(* CODESYS project DemoNov3.project
   Author: Cooper Power Systems
   Title: CoDeSys Project
   Version: 1.0.0.0
   Description: Sample Project
   Company: Cooper Power Systems LLC

Project tree, tasks and I/O mapping:
  Device : SMP SG 4000, Cooper Power Systems, LLC., order no. 
      , version 3.5.2.0
    application Application
      libraries: SmpLib, 3.5.2.0 (Cooper Power Systems); Standard, 3.5.2.0 (System)
      task Main_Task (cyclic, interval T#10ms, priority 0) calls PLC_MAIN, Tasks_10ms
      task Task_50ms (cyclic, interval t#250ms, priority 1) calls Tasks_50ms
      task Task_100ms (cyclic, interval t#100ms, priority 2) calls Tasks_100ms
      task Task_300ms (cyclic, interval t#250ms, priority 2) calls Task_300ms, POU_EXPORT
      global variables PersistentVars
      POUs/
        program PLC_MAIN [ST]
        program POU_EXPORT [ST]
        program SMP_Csys_var_AI [ST]
        program MICROGRID_MODES [ST]
        program VDC [ST]
        program SMP_Csys_var_AO [FBD]
        program LOAD_Balance [ST]
        program Load_Shed [ST]
        program SMP_OUTPUTS [FBD]
        program INIT [ST]
        program Vijay [FBD]
        program Timers [FBD]
        program PCC_CNTL [FBD]
        program Tasks_10ms [ST]
        program MICROGRID_Apps [ST]
        program Tasks_50ms [ST]
        program Tasks_100ms [ST]
        program Task_300ms [ST]
        program BRK_CNTL [ST]
        program POU_RESET [ST]
        program SMP_AO [ST]
        program TIMER_ST [ST]
        program PCC_PROTECT [ST]
        program SOC_MNGT [ST]
        program Q_Export [ST]
      function block SMP_MAP_SYMBOLS [ST]
      global variables SMP_global_symbols_declaration
      global variables Global_Variables
  function GetNumberProperty [ST]
  function GetBooleanProperty [ST]
  function GetCompany [ST]
  function GetTitle [ST]
  function GetVersionProperty [ST]
  function GetVersion [ST]
  function GetTextProperty [ST]
*)

// Device/Application/PersistentVars
VAR_GLOBAL PERSISTENT RETAIN
	PERSIST_COUNTER: DINT := 0;
	CONDITION: INT;
	GRID_APP_SELECT: INT := 0;
	ISLAND_APP_SELECT: INT := 0;
	
	// Lower frequency power limit for G1
	F_G1_L: REAL := 0;
	F_G1_H: REAL := 0;
	F_G2_L: REAL := 0;
	F_G2_H: REAL := 0;
	F_PV_L: REAL := 0;
	F_PV_H: REAL := 0;
	F_ES_L: REAL := 0;
	F_ES_H: REAL := 0;
	
	F_L9_L: REAL := 0;
	F_L9_H: REAL := 0;
	F_L10_L: REAL := 0;
	F_L10_H: REAL := 0;
	F_L11_L: REAL := 0;
	F_L11_H: REAL := 0;
	F_L15_L: REAL := 0;
	F_L15_H: REAL := 0;
	F_L16_L: REAL := 0;
	F_L16_H: REAL := 0;
	F_L20_L: REAL := 0;
	F_L20_H: REAL := 0;
	
	P_R2: REAL := 0;
	P_R3: REAL := 0;
	P_R4: REAL := 0;
	P_R5: REAL := 0;
	P_R6: REAL := 0;
	P_R7: REAL := 0;
	P_R8: REAL := 0;
	P_R9: REAL := 0;
	P_R10: REAL := 0;
	P_R11: REAL := 0;
	P_R12: REAL := 0;
	P_R13: REAL := 0;
	P_R14: REAL := 0;
	P_R15: REAL := 0;
	P_R16: REAL := 0;
	P_R17: REAL := 0;
	P_R18: REAL := 0;
	P_R19: REAL := 0;
	P_R20: REAL := 0;
	P_R21: REAL := 0;
	P_R22: REAL := 0;
	Q_R2: REAL := 0;
	Q_R3: REAL := 0;
	Q_R4: REAL := 0;
	Q_R5: REAL := 0;
	Q_R6: REAL := 0;
	Q_R7: REAL := 0;
	Q_R8: REAL := 0;
	Q_R9: REAL := 0;
	Q_R10: REAL := 0;
	Q_R11: REAL := 0;
	Q_R12: REAL := 0;
	Q_R13: REAL := 0;
	Q_R14: REAL := 0;
	Q_R15: REAL := 0;
	Q_R16: REAL := 0;
	Q_R17: REAL := 0;
	Q_R18: REAL := 0;
	Q_R19: REAL := 0;
	Q_R20: REAL := 0;
	Q_R21: REAL := 0;
	Q_R22: REAL := 0;
	StPCC: INT := 0;
	PTL_Mode1: REAL := 0;
	PTL_Mode2: REAL := 0;
	QTL_Mode1: REAL := 0;
	QTL_Mode2: REAL := 0;
//	MG_Base_P: REAL := 9.0;
//	MG_Base_Q: REAL := 5.0;
	F_BL_L: REAL := 0;
	F_BL_H: REAL := 0;
	F: REAL := 0;
	Gen1_CapW: REAL := 0;
	V_G1_L: REAL := 0;
	V_G1_H: REAL := 0;
	V_G2_L: REAL := 0;
	V_G2_H: REAL := 0;
	V_PV_L: REAL := 0;
	V_PV_H: REAL := 0;
	V_ES_L: REAL := 0;
	V_ES_H: REAL := 0;
	
	V_L9_L: REAL := 0;
	V_L9_H: REAL := 0;
	V_L10_L: REAL := 0;
	V_L10_H: REAL := 0;
	V_L11_L: REAL := 0;
	V_L11_H: REAL := 0;
	V_L15_L: REAL := 0;
	V_L15_H: REAL := 0;
	V_L16_L: REAL := 0;
	V_L16_H: REAL := 0;
	V_L20_L: REAL := 0;
	V_L20_H: REAL := 0;

	V_BL_L: REAL := 0;
	V_BL_H: REAL := 0;
	V: REAL := 0;
	Gen1_Capkvar: REAL := 0;
	Gen2_CapW: REAL := 0;
	Gen2_Capkvar: REAL := 0;
	PESS_CMD: REAL := 0;
	QESS_CMD: REAL := 0;
	BRK_PCC_CNTL: INT := 0;
	BRK_O2_CNTL: INT := 0;
	BRK_O3_CNTL: INT := 0;
	BRK_O4_CNTL: INT := 0;
	BRK_O5_CNTL: INT := 0;
	BRK_O6_CNTL: INT := 0;
	BRK_O7_CNTL: INT := 0;
	BRK_O8_CNTL: INT := 0;
	BRK_O9_CNTL: INT := 0;
	BRK_O10_CNTL: INT := 0;
	BRK_O11_CNTL: INT := 0;
	BRK_O12_CNTL: INT := 0;
	BRK_O13_CNTL: INT := 0;
	BRK_O14_CNTL: INT := 0;
	BRK_O15_CNTL: INT := 0;
	BRK_O16_CNTL: INT := 0;
	BRK_O17_CNTL: INT := 0;
	BRK_O18_CNTL: INT := 0;
	BRK_O19_CNTL: INT := 0;
	BRK_O20_CNTL: INT := 0;
	BRK_O21_CNTL: INT := 0;
	BRK_O22_CNTL: INT := 0;
	// GEN1 start/stop command
	GEN1_SS_CNTL: INT := 0;
	GEN2_SS_CNTL: INT := 0;
	ESS_SS_CNTL: INT := 0;
	PV_SS_CNTL: INT := 0;
	GEN1_MOD_sel: INT := 0;
	GEN2_MOD_sel: INT := 0;
	BAT_Enb_set: INT := 0;
	//kw//
	GEN1_kW_Out: REAL := 0;
	MG_kW_Out: REAL := 0;
	GEN2_kW_Out: REAL := 0;
	ESS_kW_Out: REAL := 0;
	PV_kW_Out: REAL := 0;
	MG_kW_Bal: REAL := 0;
	
	//kvar//
	GEN1_kVAr_Out: REAL := 0;
	MG_kVAr_Out: REAL := 0;
	GEN2_kVAr_Out: REAL := 0;
	ESS_kVAr_Out: REAL := 0;
	PV_kVAr_Out: REAL := 0;
	MG_kVAr_Bal: REAL := 0;
	
	BRKGEN1_TRIG: BOOL := 0;
	BRKGEN1_RTRIG: R_TRIG;
	BRKGEN1_FTRIG: F_TRIG;
	
	BRKGEN2_TRIG: BOOL := 0;
	BRKGEN2_RTRIG: R_TRIG;
	BRKGEN2_FTRIG: F_TRIG;
	
	BRKESS_TRIG: BOOL := 0;
	BRKESS_RTRIG: R_TRIG;
	BRKESS_FTRIG: F_TRIG;
	
	BRKPCC_TRIG: BOOL := 0;
	BRKPCC_RTRIG: R_TRIG;
	BRKPCC_FTRIG: F_TRIG;
	
	BRK2_TRIG: BOOL := 0;
	BRK2_RTRIG: R_TRIG;
	BRK2_FTRIG: F_TRIG;
	BRK3_TRIG: BOOL := 0;
	BRK3_RTRIG: R_TRIG;
	BRK3_FTRIG: F_TRIG;
	BRK4_TRIG: BOOL := 0;
	BRK4_RTRIG: R_TRIG;
	BRK4_FTRIG: F_TRIG;
	BRK5_TRIG: BOOL := 0;
	BRK5_RTRIG: R_TRIG;
	BRK5_FTRIG: F_TRIG;
	BRK6_TRIG: BOOL := 0;
	BRK6_RTRIG: R_TRIG;
	BRK6_FTRIG: F_TRIG;
	BRK7_TRIG: BOOL := 0;
	BRK7_RTRIG: R_TRIG;
	BRK7_FTRIG: F_TRIG;
	BRK8_TRIG: BOOL := 0;
	BRK8_RTRIG: R_TRIG;
	BRK8_FTRIG: F_TRIG;
	BRK9_TRIG: BOOL := 0;
	BRK9_RTRIG: R_TRIG;
	BRK9_FTRIG: F_TRIG;
	BRK10_TRIG: BOOL := 0;
	BRK10_RTRIG: R_TRIG;
	BRK10_FTRIG: F_TRIG;
	BRK11_TRIG: BOOL := 0;
	BRK11_RTRIG: R_TRIG;
	BRK11_FTRIG: F_TRIG;
	BRK12_TRIG: BOOL := 0;
	BRK12_RTRIG: R_TRIG;
	BRK12_FTRIG: F_TRIG;
	BRK13_TRIG: BOOL := 0;
	BRK13_RTRIG: R_TRIG;
	BRK13_FTRIG: F_TRIG;
	BRK14_TRIG: BOOL := 0;
	BRK14_RTRIG: R_TRIG;
	BRK14_FTRIG: F_TRIG;
	BRK15_TRIG: BOOL := 0;
	BRK15_RTRIG: R_TRIG;
	BRK15_FTRIG: F_TRIG;
	BRK16_TRIG: BOOL := 0;
	BRK16_RTRIG: R_TRIG;
	BRK16_FTRIG: F_TRIG;
	BRK17_TRIG: BOOL := 0;
	BRK17_RTRIG: R_TRIG;
	BRK17_FTRIG: F_TRIG;
	BRK18_TRIG: BOOL := 0;
	BRK18_RTRIG: R_TRIG;
	BRK18_FTRIG: F_TRIG;
	BRK19_TRIG: BOOL := 0;
	BRK19_RTRIG: R_TRIG;
	BRK19_FTRIG: F_TRIG;
	BRK20_TRIG: BOOL := 0;
	BRK20_RTRIG: R_TRIG;
	BRK20_FTRIG: F_TRIG;
	BRK21_TRIG: BOOL := 0;
	BRK21_RTRIG: R_TRIG;
	BRK21_FTRIG: F_TRIG;
	BRK22_TRIG: BOOL := 0;
	BRK22_RTRIG: R_TRIG;
	BRK22_FTRIG: F_TRIG;
	PCC_BRK_ST2: R_TRIG;
	BRK_toggle: BOOL := 0;
	//Load Shed variables
	I_Load_02: INT := 0;//Not Used
	I_Load_03: INT := 0;//Not Used
	I_Load_04: INT := 0;//Not Used
	I_Load_05: INT := 0;
	I_Load_06: INT := 0;//Not Used
	I_Load_07: INT := 0;//Not Used
	I_Load_08: INT := 0;//Not Used
	I_Load_09: INT := 0;
	I_Load_10: INT := 0;
	I_Load_11: INT := 0;
	I_Load_012: INT := 0;//Not Used
	I_Load_013: INT := 0;//Not Used
	C_Load_014: INT := 0;
	I_Load_015: INT := 0;
	I_Load_016: INT := 0;
	I_Load_017: INT := 0;//Not Used
	C_Load_018: INT := 0;
	C_Load_019: INT := 0;
	C_Load_020: INT := 0;
	C_Load_021: INT := 0;
	C_Load_022: INT := 0;
	
	
	
	
	
	
	RESET_All: BOOL := 0;
	ISLAND_CMD: BOOL := 0;
	
	
	
	
	//Export
	ERR_T: REAL := 0;
	INT_ERR: REAL := 0;
	MG_kW_Bal2: REAL := 0;
	MG_kW_Bal3: REAL := 0;
	
	GEN2_ON: BOOL := 0;
	GEN1_ON: BOOL := 0;
	ESS_ON: BOOL := 0;
	BAT_CAP: REAL := 0;
	MSTRST2: TOF;
	PCC_Delay: TON;
END_VAR

// Device/Application/SMP_global_symbols_declaration
VAR_GLOBAL
	///
	///Consumed Ai
	SPS_ADAM1_ADAM_AI_3: AI_IN;
	SPS_ADAM1_ADAM_AI_5: AI_IN;
	SPS_GEN1_METMMXU1HzInstMag: AI_IN;
	SPS_GEN1_METMMXU1TotVArInstMag: AI_IN;
	SPS_GEN1_METMMXU1TotWInstMag: AI_IN;
	SPS_PCS_drv1_Iq_ref: AI_IN;
	SPS_SELG_METYMMXU2HzInstMag: AI_IN;
	SPS_SELG_METYMMXU2HzMag: AI_IN;
	SPS_SELG_METYMMXU2PhVPhsAIMag: AI_IN;
	SPS_SELG_METYMMXU2PhVPhsAMag: AI_IN;
	SPS_SELG_METYMMXU2TotVArInstMag: AI_IN;
	SPSSELG_METYMMXU2TotVArMag: AI_IN;
	SPSSELG_METYMMXU2TotWInstMag: AI_IN;
	SPS_SELG_METYMMXU2TotWMag: AI_IN;
	///
	///Consumed Ao
	SPS_PCS_INV1_FB2_POWDEL_INS: AO_IN;
	SPS_PCS_INV1_FB3_POWDEL_INS: AO_IN;
END_VAR

// Device/Application/Global_Variables
VAR_GLOBAL

	
PCC_BRK_ST: DINT := 0;    // 1 = BRK_Closed  0 = BRK_Open
	MIN_CLK: BOOL;
	HR_CLK: BOOL;
	Mode1_CNTR_flg: BOOL := 0;
	RUN_MIN: INT := 0;
	PPCC_CMD: REAL := 0;
	QPCC_CMD: REAL := 0;
	TMR_MIN_1: TON;
	Mode1_CNTR_1: CTU;
	TMR1_1: TON;
	TMRs_1: TON;
	Fretest: DINT := 0;
	AO_TGL_1: TON;
	AO_TGL_2: TON;
	EXP_CMD: BOOL := 0;
	Trig3: INT := 0;
	Trig4: BOOL := 0;
END_VAR
VAR_GLOBAL RETAIN
	Adam_UPC: CTU;
	T_2 : BOOL;
	T_1 : BOOL;
	ON_OFF_SW: INT;
	OUT_Visualisation: BOOL := 0;
	SET5: BOOL;
	B_Switch: BOOL := 0;
	DRV1_Cmd_Data: DINT := 0;
	DRV2_Cmd_Data: DINT := 0;
	Real_P1: DINT := 0;
	Real_P2: DINT := 0;
	SPS_Rreal_Pw: DINT := 0;
	React_P1: DINT := 0;
	React_P2: DINT := 0;
	SPS_Reactive_Pw: DINT := 0;
	PTL: REAL := 0;
	QTL: REAL := 0;
	PT: REAL := 0;
	QT: REAL := 0;
	CPG1: REAL := 10;
	CPG2: REAL := 20;
	PG1_CMD: REAL;
	PG2_CMD: REAL := 0;
	
	QG1_CMD: REAL := 0;
	QG2_CMD: REAL := 0;
	
	QG1_CMD_A: REAL := 0;
	QG2_CMD_A: REAL := 0;
	
	QG1_CMD_B: REAL := 0;
	QG2_CMD_B: REAL := 0;
	
	
	CQG1: REAL := 10;
	CQG2: REAL := 20;
	MODE: INT := 0;
	MSTRST: R_TRIG;
	Trig: BOOL := 1;
	Load_Cntr: INT := 0;
	GEN1_toggle: BOOL := 0;
	GEN2_toggle: BOOL := 0;
	ESS_toggle: BOOL := 0;
	
	///Timing
	EXP_STRT1 : INT := 5;
	EXP_STRT2 : INT := 20;
	EXP_END : INT := 35;
	ISL_STRT : INT := 36;
	ISL_END : INT := 50;
	
	MG_Base_P: REAL := 9.0;
	MG_Base_Q: REAL := 5.0;
	
END_VAR

// Device/Application/POUs/PLC_MAIN
PROGRAM PLC_MAIN

VAR
	CODESYS_INIT: BOOL := FALSE;
	CODESYS_MAP: BOOL := FALSE;
	SmpMapSymbols : SMP_MAP_SYMBOLS;
	test: INT := 0;
	test1: INT := 0;
END_VAR

(* 	Cooper Power Systems LLC
	SoftPLC Sample project
	Version 1.0, January 2013
	
	This sample is provided "as is" to reduce the user's learning curve about CoDeSys integration with the SMP Gateway. 
	Cooper Power Systems cannot be held responsible in any situation resulting from the use of this sample program.

	Currently, the SMP Gateway runtime can only run one application at a time.
    This application must be named "Application".
	This application can be developped in any IEC 611l31-3 language.

	------------- IMPORTANT (begin)------------- 
	SMP Config automatically generates a PLCopenXML file that contains the SMP_MAP_SYMBOLS function block
    and the SMP_global_symbols_declaration global variable list. When the configuration of the SoftPLC component is changed in
    SMP Config, the content of this file must then be used to update the application.

	
	To update the application with the latest version of the PLCopenXML file, follow those steps:
	
	1. In the left pane, expand the project tree and select the "Application" branch under "PLC Logic".
	2. From the "Project" menu, choose "Import PLCopenXML"
	3. Select the XML file created by SMP Config. 
		The file is under My Documents or Documents/SMP Manager/Config Files/CoDeSys_TmpEdit. 
		The filename syntax is: the SMP Config settings filename + the Soft PLC instance name + "PLCopenXML.xml".
	4.  In the "Import PLCopenXML" window, just click "Open"; the two SMP-Gateway-related items are already selected.
	5. In the next window, select option 4 "Replace the existing object. Do the same for all subsequent conflicts."
	6. You ready to rebuild the application. 

	------------- IMPORTANT (end)------------- 
*)

(* 	The code inside this IF block must be executed first, ONLY once. *)
IF (SMF_CANMAPPLC(0) AND CODESYS_INIT = FALSE) THEN

	(*  Specify basic information about this application.
		Update according to your own application requirements and functionalities. *)
	SMF_INITPLC ('Application Name is Sample',  'Author is Cooper Power Systems, LLC', 'Description is a sample program',  '1.0', LIBVERSION, T#10S);

	(* 	Add a log entry indicating that the application is starting up.
		Update as required; you can also add additional SMF_LOG function call if you want *)
	SMF_LOG(TRUE, LOG_STARTUP,'SoftPLC application is starting');
	
	(* 	SMP_Config auto-generated symbol mapping.
	   	At runtime, an exception will be thrown if there is an error. 
	   	Use SMP Log and SMP Stats to get details about the error. 
		DO NOT DELETE THIS FUNCTION CALL. *)
	SmpMapSymbols();
			
	(* 	Update the initialization flag to indicates that initialization is complete.
		DO NOT DELETE THIS LINE OF CODE. *)
	CODESYS_INIT:=TRUE;
	//INIT();	
	test := test+1;
	
ELSE
	(* The code inside this IF block must be executed ONLY once, when the symbol mapping was successful. *)
	IF (SMF_CANSTARTPLC(0) AND CODESYS_MAP = FALSE) THEN
	
		(*  Initialize the output points synbols so they can accept control requests. 	
			Change/update as required. *)
		//( B:=0, Q:=0, DIS:= FALSE, END:=FALSE );
		//( I:= 0, Q:=0, DIS:= FALSE, END:=FALSE );
		//( F:= 0.0, Q:=0 );
			
		(* 	Examples on how to write an entry into each different log.
			Change/update as required. *) 
		SMF_LOG(TRUE, LOG_APPLICATION, 'Application Log: Example PLC');
		SMF_LOG(TRUE, LOG_COMMAND,'Control Log: Example PLC');
		SMF_LOG(TRUE, LOG_FILE,'File Log: Example PLC');
		SMF_LOG(TRUE, LOG_PROTOCOL,'Protocol Log: Example PLC');
		SMF_LOG(TRUE, LOG_SECURITY,'Security Log: Example PLC');
	
		(* 	Examples on how to write to each statistic field.
			Change/update as required. *)
		SMF_STAT(TRUE, STAT_USER1, '0'); 	(* BO CMND counter *)
		SMF_STAT(TRUE, STAT_USER2, '0'); 	(* AO CMND counter *)
		SMF_STAT(TRUE, STAT_USER3, 'No Used');
		SMF_STAT(TRUE, STAT_USER4, 'No Used');
		SMF_STAT(TRUE, STAT_USER5, 'No Used');
		SMF_STAT(TRUE, STAT_USER6, 'No Used');
		SMF_STAT(TRUE, STAT_USER7, 'No Used');
		SMF_STAT(TRUE, STAT_USER8, 'No Used');
		SMF_STAT(TRUE, STAT_USER9, 'No Used');
		SMF_STAT(TRUE, STAT_USER10, 'No Used');
		SMF_STAT(TRUE, STAT_USER11, 'No Used');
		SMF_STAT(TRUE, STAT_USER12, 'No Used');
		SMF_STAT(TRUE, STAT_USER13, 'No Used');
		SMF_STAT(TRUE, STAT_USER14, 'No Used');
		SMF_STAT(TRUE, STAT_USER15, 'No Used');
		SMF_STAT(TRUE, STAT_USER16, 'No Used');
	
		(* 	Add a log entry to indicate that the SoftPLC application was started successfully.
			Change/update as required. *)
		SMF_LOG(TRUE, LOG_STARTUP,'SoftPLC application is started.');
	
		(* 	Always re-enable local control operation
			This is specific to sample project: REMOVE IT FROM YOUR OWN APPLICATION *)	
		//( CMD:=BO_CMD_OPEN , ON:=T#0S , OFF:=T#0S , RPT:=0 , OP:=1 );
		//INPUT_BO_SetLocalControl( OP:=0 );
		
		(* 	Symbol mapping is completed and all points were initialized.
			DO NOT DELETE THIS LINE OF CODE. *)
		CODESYS_MAP:=TRUE;
	
	(* The code inside this IF block must be executed at each cycle, once INIT is completed. *)
	ELSIF (SMF_CANSTARTPLC(0) AND CODESYS_MAP = TRUE) THEN
	
		(* 	Call the main application coded in Structured Text.
			You can call any of your programs coded in any IEC 61131-3 language here.
			Change/update as required. *)
	//	ST_PROGRAM();
	//	Vijay();
	//	Timers();
		IF MSTRST2.Q = 1 THEN
			POU_RESET();
			test1 := test1+1;
		END_IF
	END_IF
END_IF

END_PROGRAM

// Device/Application/SMP_MAP_SYMBOLS
FUNCTION_BLOCK SMP_MAP_SYMBOLS

	(* Auto-generated by SMP Config, do not modify *)

	(* Subscribed points mapping *)
	SMF_MAP_AI_IN(ADR(SPS_ADAM1_ADAM_AI_3), 'ADAM1_ADAM_AI_3', 0);
	SMF_MAP_AI_IN(ADR(SPS_ADAM1_ADAM_AI_5), 'ADAM1_ADAM_AI_5', 0);
	SMF_MAP_AI_IN(ADR(SPS_GEN1_METMMXU1HzInstMag), 'GEN1_METMMXU1HzInstMag', 0);
	SMF_MAP_AI_IN(ADR(SPS_GEN1_METMMXU1TotVArInstMag), 'GEN1_METMMXU1TotVArInstMag', 0);
	SMF_MAP_AI_IN(ADR(SPS_GEN1_METMMXU1TotWInstMag), 'GEN1_METMMXU1TotWInstMag', 0);
	SMF_MAP_AI_IN(ADR(SPS_PCS_drv1_Iq_ref), 'PCS_drv1_Iq_ref', 0);
	SMF_MAP_AI_IN(ADR(SPS_SELG_METYMMXU2HzInstMag), 'SELG_METYMMXU2HzInstMag', 0);
	SMF_MAP_AI_IN(ADR(SPS_SELG_METYMMXU2HzMag), 'SELG_METYMMXU2HzMag', 0);
	SMF_MAP_AI_IN(ADR(SPS_SELG_METYMMXU2PhVPhsAIMag), 'SELG_METYMMXU2PhVPhsAIMag', 0);
	SMF_MAP_AI_IN(ADR(SPS_SELG_METYMMXU2PhVPhsAMag), 'SELG_METYMMXU2PhVPhsAMag', 0);
	SMF_MAP_AI_IN(ADR(SPS_SELG_METYMMXU2TotVArInstMag), 'SELG_METYMMXU2TotVArInstMag', 0);
	SMF_MAP_AI_IN(ADR(SPSSELG_METYMMXU2TotVArMag), 'SELG_METYMMXU2TotVArMag', 0);
	SMF_MAP_AI_IN(ADR(SPSSELG_METYMMXU2TotWInstMag), 'SELG_METYMMXU2TotWInstMag', 0);
	SMF_MAP_AI_IN(ADR(SPS_SELG_METYMMXU2TotWMag), 'SELG_METYMMXU2TotWMag', 0);

	SMF_MAP_AO_IN(ADR(SPS_PCS_INV1_FB2_POWDEL_INS), 'PCS_INV1_FB2_POWDEL_INS', 0);
	SMF_MAP_AO_IN(ADR(SPS_PCS_INV1_FB3_POWDEL_INS), 'PCS_INV1_FB3_POWDEL_INS', 0);

END_FUNCTION_BLOCK

// Device/Application/POUs/INIT
PROGRAM INIT
VAR
END_VAR

//--------------Initialization of System variables------------//
BRK_PCC_CNTL := 1;
BRK_O2_CNTL := 1;
BRK_O3_CNTL := 1;
BRK_O4_CNTL := 1;
BRK_O5_CNTL := 1;
BRK_O6_CNTL := 1;
BRK_O7_CNTL := 1;
BRK_O8_CNTL := 1;
BRK_O9_CNTL := 1;
BRK_O10_CNTL := 1;
BRK_O11_CNTL := 1;
BRK_O12_CNTL := 1;
BRK_O13_CNTL := 1;
BRK_O14_CNTL := 1;
BRK_O15_CNTL := 1;
BRK_O16_CNTL := 1;
BRK_O17_CNTL := 1;
BRK_O18_CNTL := 1;
BRK_O19_CNTL := 1;
BRK_O20_CNTL := 1;
BRK_O21_CNTL := 1;
BRK_O22_CNTL := 1;
//--------------------------------------------------------------//

//--------------Initialization of System controls start/stop------------//
GEN1_SS_CNTL := 1;
GEN2_SS_CNTL := 1;

ESS_SS_CNTL := 1;

PV_SS_CNTL := 1;
//--------------------------------------------------------------//

//--------------Initialization of Device Modes of operation------------//
GEN1_MOD_sel := 1;
GEN2_MOD_sel := 1;

BAT_Enb_set := 1;
//--------------------------------------------------------------//

//-------Mode1_Counter_Flag ----------------------//
Mode1_CNTR_flg := 1;  //refrence in timer pou for HR clk
RUN_MIN := 0;
MIN_CLK := 0;
HR_CLK := 0;
//------------------------------------------------//

//--INIT all Breakers AO--//

BRK_toggle := FALSE; 
BRK_CNTL();
RESET_All := 1;
//POU_RESET();
//------------------------//

END_PROGRAM

// Device/Application/POUs/BRK_CNTL
PROGRAM BRK_CNTL
VAR
	test: INT := 0;
	test2: INT := 0;
	BRK2_Trig2: BOOL := 0;
END_VAR

//-----------Below all Interruptable loads are controlled by expot mode-----------//
IF (NOT ISLAND_CMD) THEN   // Export Mode 
	I_Load_05 := 1;
	I_Load_09 := 1;
	I_Load_10 := 1;
	I_Load_11 := 1;
	I_Load_015 := 1;
	I_Load_016 := 1;
	
	C_Load_014 := 1;
	C_Load_018 := 1;
	C_Load_019 := 1;
	C_Load_020 := 1;
	C_Load_021 := 1;
	C_Load_022 := 1;
	
END_IF 
//--------------------------------------------------------------------------------//

BRKPCC_RTRIG(CLK := INT_TO_BOOL(PersistentVars.BRK_PCC_CNTL ) AND BRK_toggle);
BRKPCC_FTRIG(CLK := INT_TO_BOOL(PersistentVars.BRK_PCC_CNTL ) AND BRK_toggle); 
 IF ((BRKPCC_RTRIG.Q = TRUE) OR (BRKPCC_FTRIG.Q = TRUE)) THEN
	BRKPCC_TRIG := TRUE;
	test := test+1;
 ELSE 
	BRKPCC_TRIG := FALSE;
	test2 := test2+1;
 END_IF
SMP_global_symbols_declaration.C_PCC1_XCBR1RmtCtrlSetVal(ISET := PersistentVars.BRK_PCC_CNTL , IOP:=Trig);


///---Breaker ON/OFF Commands----//
IF PersistentVars.BRK_PCC_CNTL = 0 THEN
	PersistentVars.BRK_O2_CNTL := 0;
ELSE
	PersistentVars.BRK_O2_CNTL := 0;
END_IF
IF PersistentVars.BRK_PCC_CNTL = 0 THEN
	PersistentVars.BRK_O3_CNTL := 0;
ELSE
	PersistentVars.BRK_O3_CNTL := 0;
END_IF
IF PersistentVars.BRK_PCC_CNTL = 0 THEN
	PersistentVars.BRK_O4_CNTL := 0;
ELSE
	PersistentVars.BRK_O4_CNTL := 0;
END_IF

IF PersistentVars.BRK_PCC_CNTL = 0  THEN
	PersistentVars.BRK_O5_CNTL := 0;
ELSIF I_Load_05 = 1 THEN
	PersistentVars.BRK_O5_CNTL := 0;
	ELSE
	PersistentVars.BRK_O5_CNTL := 1;
END_IF
IF PersistentVars.BRK_PCC_CNTL = 0 THEN
	PersistentVars.BRK_O6_CNTL := 0;
ELSE
	PersistentVars.BRK_O6_CNTL := 0;
END_IF
IF (PersistentVars.BRK_PCC_CNTL = 0 AND PCC_Delay.Q) OR ISLAND_CMD THEN
	PersistentVars.BRK_O7_CNTL := 0;
ELSE
	PersistentVars.BRK_O7_CNTL := 1;
END_IF
IF (PersistentVars.BRK_PCC_CNTL = 0 AND PCC_Delay.Q) OR ISLAND_CMD THEN
	PersistentVars.BRK_O8_CNTL := 0;
ELSE
	PersistentVars.BRK_O8_CNTL := 1;
END_IF
IF PersistentVars.BRK_PCC_CNTL = 0 THEN
	PersistentVars.BRK_O9_CNTL := 0;
ELSIF I_Load_09 = 1 THEN
	PersistentVars.BRK_O9_CNTL := 0;
	ELSE
	PersistentVars.BRK_O9_CNTL := 1;
END_IF
IF PersistentVars.BRK_PCC_CNTL = 0 THEN
	PersistentVars.BRK_O10_CNTL := 0;
ELSIF I_Load_10 = 1 THEN
	PersistentVars.BRK_O10_CNTL := 0;
	ELSE
	PersistentVars.BRK_O10_CNTL := 1;
END_IF
IF PersistentVars.BRK_PCC_CNTL = 0 THEN
	PersistentVars.BRK_O11_CNTL := 0;
ELSIF I_Load_11 = 1 THEN
	PersistentVars.BRK_O11_CNTL := 0;
	ELSE
	PersistentVars.BRK_O11_CNTL := 1;
END_IF
IF PersistentVars.BRK_PCC_CNTL = 0 THEN
	PersistentVars.BRK_O12_CNTL := 0;
ELSE
	PersistentVars.BRK_O12_CNTL := 0;
END_IF
IF PersistentVars.BRK_PCC_CNTL = 0 THEN
	PersistentVars.BRK_O13_CNTL := 0;
ELSE
	PersistentVars.BRK_O13_CNTL := 0;
END_IF
IF PersistentVars.BRK_PCC_CNTL = 0 THEN
	PersistentVars.BRK_O14_CNTL := 0;
ELSIF C_Load_014 = 1 THEN
	PersistentVars.BRK_O14_CNTL := 0;
	ELSE
	PersistentVars.BRK_O14_CNTL := 1;
END_IF
IF PersistentVars.BRK_PCC_CNTL = 0 THEN
	PersistentVars.BRK_O15_CNTL := 0;
ELSIF I_Load_015 = 1 THEN
	PersistentVars.BRK_O15_CNTL := 0;
	ELSE
	PersistentVars.BRK_O15_CNTL := 1;
END_IF
IF PersistentVars.BRK_PCC_CNTL = 0 THEN
	PersistentVars.BRK_O16_CNTL := 0;
ELSIF I_Load_016 = 1 THEN
	PersistentVars.BRK_O16_CNTL := 0;
	ELSE
	PersistentVars.BRK_O16_CNTL := 1;
END_IF
IF (PersistentVars.BRK_PCC_CNTL = 0  OR (RUN_MIN >= C_AF_ISL_STRT.I))THEN  // ** Check if GEN1 is not ON
	PersistentVars.BRK_O17_CNTL := 0;
ELSE
	PersistentVars.BRK_O17_CNTL := 1;
END_IF
IF PersistentVars.BRK_PCC_CNTL = 0 THEN
	PersistentVars.BRK_O18_CNTL := 0;
	ELSIF C_Load_018 = 1 THEN
	PersistentVars.BRK_O18_CNTL := 0;
ELSE
	PersistentVars.BRK_O18_CNTL := 1;
END_IF
IF PersistentVars.BRK_PCC_CNTL = 0 THEN
	PersistentVars.BRK_O19_CNTL := 0;
	ELSIF C_Load_019 = 1 THEN
	PersistentVars.BRK_O19_CNTL := 0;
ELSE
	PersistentVars.BRK_O19_CNTL := 1;
END_IF
IF PersistentVars.BRK_PCC_CNTL = 0 THEN
	PersistentVars.BRK_O20_CNTL := 0;
ELSIF C_Load_020 = 1 THEN
	PersistentVars.BRK_O20_CNTL := 0;
	ELSE
	PersistentVars.BRK_O20_CNTL := 1;	
END_IF
IF PersistentVars.BRK_PCC_CNTL = 0 THEN
	PersistentVars.BRK_O21_CNTL := 0;
	ELSIF C_Load_021 = 1 THEN
	PersistentVars.BRK_O21_CNTL := 0;
ELSE
	PersistentVars.BRK_O21_CNTL := 1;
END_IF
IF PersistentVars.BRK_PCC_CNTL = 0 THEN
	PersistentVars.BRK_O22_CNTL := 0;
	ELSIF C_Load_022 = 1 THEN
	PersistentVars.BRK_O22_CNTL := 0;
ELSE
	PersistentVars.BRK_O22_CNTL := 1;
END_IF
//----------------//

BRK2_RTRIG(CLK := INT_TO_BOOL(PersistentVars.BRK_O2_CNTL ) AND BRK_toggle);
BRK2_FTRIG(CLK := INT_TO_BOOL(PersistentVars.BRK_O2_CNTL ) AND BRK_toggle); 
 IF ((BRK2_RTRIG.Q = TRUE) OR (BRK2_FTRIG.Q = TRUE)) THEN
	BRK2_TRIG := TRUE;
	test := test+1;
 ELSE 
	BRK2_TRIG := FALSE;
	test2 := test2+1;
 END_IF
SMP_global_symbols_declaration.C_BRKS_XCBR2Pos_CtrlSetVal(ISET := PersistentVars.BRK_O2_CNTL , IOP:=BRK2_TRIG);


BRK3_RTRIG(CLK :=INT_TO_BOOL(PersistentVars.BRK_O3_CNTL ) AND BRK_toggle);
BRK3_FTRIG(CLK :=INT_TO_BOOL(PersistentVars.BRK_O3_CNTL ) AND BRK_toggle);  
 IF BRK3_RTRIG.Q = 1 OR BRK3_FTRIG.Q = 1 THEN
	BRK3_TRIG := 1;
 ELSE 
	BRK3_TRIG := 0;
 END_IF
SMP_global_symbols_declaration.C_BRKS_XCBR3Pos_CtrlSetVal(ISET := PersistentVars.BRK_O3_CNTL , IOP:=BRK3_TRIG);


BRK4_RTRIG(CLK :=INT_TO_BOOL(PersistentVars.BRK_O4_CNTL ) AND BRK_toggle);
BRK4_FTRIG(CLK :=INT_TO_BOOL(PersistentVars.BRK_O4_CNTL ) AND BRK_toggle);  
 IF BRK4_RTRIG.Q = 1 OR BRK4_FTRIG.Q = 1 THEN
	BRK4_TRIG := 1;
 ELSE 
	BRK4_TRIG := 0;
 END_IF
SMP_global_symbols_declaration.C_BRKS_XCBR4Pos_CtrlSetVal(ISET := PersistentVars.BRK_O4_CNTL , IOP:=BRK4_TRIG);


BRK5_RTRIG(CLK :=INT_TO_BOOL(PersistentVars.BRK_O5_CNTL ) AND BRK_toggle);
BRK5_FTRIG(CLK :=INT_TO_BOOL(PersistentVars.BRK_O5_CNTL ) AND BRK_toggle);  
 IF BRK5_RTRIG.Q = 1 OR BRK5_FTRIG.Q = 1 THEN
	BRK5_TRIG := 1;
 ELSE 
	BRK5_TRIG := 0;
 END_IF
SMP_global_symbols_declaration.C_BRKS_XCBR5Pos_CtrlSetVal(ISET := PersistentVars.BRK_O5_CNTL , IOP:=BRK5_TRIG);


BRK6_RTRIG(CLK :=INT_TO_BOOL(PersistentVars.BRK_O6_CNTL ) AND BRK_toggle);
BRK6_FTRIG(CLK :=INT_TO_BOOL(PersistentVars.BRK_O6_CNTL ) AND BRK_toggle);  
 IF BRK6_RTRIG.Q = 1 OR BRK6_FTRIG.Q = 1 THEN
	BRK6_TRIG := 1;
 ELSE 
	BRK6_TRIG := 0;
 END_IF
SMP_global_symbols_declaration.C_BRKS_XCBR6Pos_CtrlSetVal(ISET := PersistentVars.BRK_O6_CNTL , IOP:=BRK6_TRIG);


BRK7_RTRIG(CLK :=INT_TO_BOOL(PersistentVars.BRK_O7_CNTL ) AND BRK_toggle);
BRK7_FTRIG(CLK :=INT_TO_BOOL(PersistentVars.BRK_O7_CNTL ) AND BRK_toggle);  
 IF BRK7_RTRIG.Q = 1 OR BRK7_FTRIG.Q = 1 THEN
	BRK7_TRIG := 1;
 ELSE 
	BRK7_TRIG := 0;
 END_IF
SMP_global_symbols_declaration.C_BRKS_XCBR7Pos_CtrlSetVal(ISET := PersistentVars.BRK_O7_CNTL , IOP:=BRK7_TRIG);


BRK8_RTRIG(CLK :=INT_TO_BOOL(PersistentVars.BRK_O8_CNTL ) AND BRK_toggle);
BRK8_FTRIG(CLK :=INT_TO_BOOL(PersistentVars.BRK_O8_CNTL ) AND BRK_toggle);  
 IF BRK8_RTRIG.Q = 1 OR BRK8_FTRIG.Q = 1 THEN
	BRK8_TRIG := 1;
 ELSE 
	BRK8_TRIG := 0;
 END_IF
SMP_global_symbols_declaration.C_BRKS_XCBR8Pos_CtrlSetVal(ISET := PersistentVars.BRK_O8_CNTL , IOP:=BRK8_TRIG);


BRK9_RTRIG(CLK :=INT_TO_BOOL(PersistentVars.BRK_O9_CNTL ) AND BRK_toggle);
BRK9_FTRIG(CLK :=INT_TO_BOOL(PersistentVars.BRK_O9_CNTL ) AND BRK_toggle);  
 IF BRK9_RTRIG.Q = 1 OR BRK9_FTRIG.Q = 1 THEN
	BRK9_TRIG := 1;
 ELSE 
	BRK9_TRIG := 0;
 END_IF
SMP_global_symbols_declaration.C_BRKS_XCBR9Pos_CtrlSetVal(ISET := PersistentVars.BRK_O9_CNTL , IOP:=BRK9_TRIG);


BRK10_RTRIG(CLK :=INT_TO_BOOL(PersistentVars.BRK_O10_CNTL ) AND BRK_toggle);
BRK10_FTRIG(CLK :=INT_TO_BOOL(PersistentVars.BRK_O10_CNTL ) AND BRK_toggle);  
 IF BRK10_RTRIG.Q = 1 OR BRK10_FTRIG.Q = 1 THEN
	BRK10_TRIG := 1;
 ELSE 
	BRK10_TRIG := 0;
 END_IF
SMP_global_symbols_declaration.C_BRKS_XCBR10Pos_CtrlSetVal(ISET := PersistentVars.BRK_O10_CNTL , IOP:=BRK10_TRIG);


BRK11_RTRIG(CLK :=INT_TO_BOOL(PersistentVars.BRK_O11_CNTL ) AND BRK_toggle);
BRK11_FTRIG(CLK :=INT_TO_BOOL(PersistentVars.BRK_O11_CNTL ) AND BRK_toggle);  
 IF BRK11_RTRIG.Q = 1 OR BRK11_FTRIG.Q = 1 THEN
	BRK11_TRIG := 1;
 ELSE 
	BRK11_TRIG := 0;
 END_IF
SMP_global_symbols_declaration.C_BRKS_XCBR11Pos_CtrlSetVal(ISET := PersistentVars.BRK_O11_CNTL , IOP:=BRK11_TRIG);


BRK12_RTRIG(CLK :=INT_TO_BOOL(PersistentVars.BRK_O12_CNTL ) AND BRK_toggle);
BRK12_FTRIG(CLK :=INT_TO_BOOL(PersistentVars.BRK_O12_CNTL ) AND BRK_toggle);  
 IF BRK12_RTRIG.Q = 1 OR BRK12_FTRIG.Q = 1 THEN
	BRK12_TRIG := 1;
 ELSE 
	BRK12_TRIG := 0;
 END_IF
SMP_global_symbols_declaration.C_BRKS_XCBR12Pos_CtrlSetVal(ISET := PersistentVars.BRK_O12_CNTL , IOP:=BRK12_TRIG);


BRK13_RTRIG(CLK :=INT_TO_BOOL(PersistentVars.BRK_O13_CNTL ) AND BRK_toggle);
BRK13_FTRIG(CLK :=INT_TO_BOOL(PersistentVars.BRK_O13_CNTL ) AND BRK_toggle);  
 IF BRK13_RTRIG.Q = 1 OR BRK13_FTRIG.Q = 1 THEN
	BRK13_TRIG := 1;
 ELSE 
	BRK13_TRIG := 0;
 END_IF
SMP_global_symbols_declaration.C_BRKS_XCBR13Pos_CtrlSetVal(ISET := PersistentVars.BRK_O13_CNTL , IOP:=BRK13_TRIG);


BRK14_RTRIG(CLK :=INT_TO_BOOL(PersistentVars.BRK_O14_CNTL ) AND BRK_toggle);
BRK14_FTRIG(CLK :=INT_TO_BOOL(PersistentVars.BRK_O14_CNTL ) AND BRK_toggle);  
 IF BRK14_RTRIG.Q = 1 OR BRK14_FTRIG.Q = 1 THEN
	BRK14_TRIG := 1;
 ELSE 
	BRK14_TRIG := 0;
 END_IF
SMP_global_symbols_declaration.C_BRKS_XCBR14Pos_CtrlSetVal(ISET := PersistentVars.BRK_O14_CNTL , IOP:=BRK14_TRIG);


BRK15_RTRIG(CLK :=INT_TO_BOOL(PersistentVars.BRK_O15_CNTL ) AND BRK_toggle);
BRK15_FTRIG(CLK :=INT_TO_BOOL(PersistentVars.BRK_O15_CNTL ) AND BRK_toggle);  
 IF BRK15_RTRIG.Q = 1 OR BRK15_FTRIG.Q = 1 THEN
	BRK15_TRIG := 1;
 ELSE 
	BRK15_TRIG := 0;
 END_IF
SMP_global_symbols_declaration.C_BRKS_XCBR15Pos_CtrlSetVal(ISET := PersistentVars.BRK_O15_CNTL , IOP:=BRK15_TRIG);



BRK16_RTRIG(CLK :=INT_TO_BOOL(PersistentVars.BRK_O16_CNTL ) AND BRK_toggle);
BRK16_FTRIG(CLK :=INT_TO_BOOL(PersistentVars.BRK_O16_CNTL ) AND BRK_toggle);  
 IF BRK16_RTRIG.Q = 1 OR BRK16_FTRIG.Q = 1 THEN
	BRK16_TRIG := 1;
 ELSE 
	BRK16_TRIG := 0;
 END_IF
SMP_global_symbols_declaration.C_BRKS_XCBR16Pos_CtrlSetVal(ISET := PersistentVars.BRK_O16_CNTL , IOP:=BRK16_TRIG);


BRK17_RTRIG(CLK :=INT_TO_BOOL(PersistentVars.BRK_O17_CNTL ) AND BRK_toggle);
BRK17_FTRIG(CLK :=INT_TO_BOOL(PersistentVars.BRK_O17_CNTL ) AND BRK_toggle);  
 IF BRK17_RTRIG.Q = 1 OR BRK17_FTRIG.Q = 1 THEN
	BRK17_TRIG := 1;
 ELSE 
	BRK17_TRIG := 0;
 END_IF
SMP_global_symbols_declaration.C_BRKS_XCBR17Pos_CtrlSetVal(ISET := PersistentVars.BRK_O17_CNTL , IOP:=BRK17_TRIG);


BRK18_RTRIG(CLK :=INT_TO_BOOL(PersistentVars.BRK_O18_CNTL ) AND BRK_toggle);
BRK18_FTRIG(CLK :=INT_TO_BOOL(PersistentVars.BRK_O18_CNTL ) AND BRK_toggle);  
 IF BRK18_RTRIG.Q = 1 OR BRK18_FTRIG.Q = 1 THEN
	BRK18_TRIG := 1;
 ELSE 
	BRK18_TRIG := 0;
 END_IF
SMP_global_symbols_declaration.C_BRKS_XCBR18Pos_CtrlSetVal(ISET := PersistentVars.BRK_O18_CNTL , IOP:=BRK18_TRIG);


BRK19_RTRIG(CLK :=INT_TO_BOOL(PersistentVars.BRK_O19_CNTL ) AND BRK_toggle);
BRK19_FTRIG(CLK :=INT_TO_BOOL(PersistentVars.BRK_O19_CNTL ) AND BRK_toggle);
 IF BRK19_RTRIG.Q = 1 OR BRK19_FTRIG.Q = 1 THEN
	BRK19_TRIG := 1;
 ELSE 
	BRK19_TRIG := 0;
 END_IF
SMP_global_symbols_declaration.C_BRKS_XCBR19Pos_CtrlSetVal(ISET := PersistentVars.BRK_O19_CNTL , IOP:=BRK19_TRIG);



BRK20_RTRIG(CLK :=INT_TO_BOOL(PersistentVars.BRK_O20_CNTL ) AND BRK_toggle);
BRK20_FTRIG(CLK :=INT_TO_BOOL(PersistentVars.BRK_O20_CNTL ) AND BRK_toggle);  
 IF BRK20_RTRIG.Q = 1 OR BRK20_FTRIG.Q = 1 THEN
	BRK20_TRIG := 1;
 ELSE 
	BRK20_TRIG := 0;
 END_IF
SMP_global_symbols_declaration.C_BRKS_XCBR20Pos_CtrlSetVal(ISET := PersistentVars.BRK_O20_CNTL , IOP:=BRK20_TRIG);


BRK21_RTRIG(CLK :=INT_TO_BOOL(PersistentVars.BRK_O21_CNTL ) AND BRK_toggle);
BRK21_FTRIG(CLK :=INT_TO_BOOL(PersistentVars.BRK_O21_CNTL ) AND BRK_toggle);  
 IF BRK21_RTRIG.Q = 1 OR BRK21_FTRIG.Q = 1 THEN
	BRK21_TRIG := 1;
 ELSE 
	BRK21_TRIG := 0;
 END_IF
SMP_global_symbols_declaration.C_BRKS_XCBR21Pos_CtrlSetVal(ISET := PersistentVars.BRK_O21_CNTL , IOP:=BRK21_TRIG);


BRK22_RTRIG(CLK :=INT_TO_BOOL(PersistentVars.BRK_O22_CNTL ) AND BRK_toggle);
BRK22_FTRIG(CLK :=INT_TO_BOOL(PersistentVars.BRK_O22_CNTL ) AND BRK_toggle);  
 IF BRK22_RTRIG.Q = 1 OR BRK22_FTRIG.Q = 1 THEN
	BRK22_TRIG := 1;
 ELSE 
	BRK22_TRIG := 0;
 END_IF
SMP_global_symbols_declaration.C_BRKS_XCBR22Pos_CtrlSetVal(ISET := PersistentVars.BRK_O22_CNTL , IOP:=BRK22_TRIG);


BRK_toggle := TRUE; 	
//END_IF

END_PROGRAM

// Device/Application/POUs/POU_RESET
PROGRAM POU_RESET
VAR
	test1: INT := 0;
END_VAR


	PersistentVars.GEN1_SS_CNTL := 0;
	PersistentVars.GEN2_SS_CNTL := 0;
	PersistentVars.ESS_SS_CNTL := 0;
	PersistentVars.PV_SS_CNTL := 0;
	RUN_MIN := 0;
	GEN1_kW_Out := 0;
	GEN2_kW_Out := 0;
	ESS_kW_Out := 0;
	GEN1_kVAr_Out := 0;
	GEN2_kVAr_Out :=0 ;
	ESS_kVAr_Out := 0;
	MG_kW_Out := 0;
	test1 := test1+1;
	ERR_T := 0;
	INT_ERR := 0;
	MG_kW_Bal2 := 0;
	MG_kW_Bal3 := 0;
	MG_kW_Bal := 0;
	ISLAND_CMD := FALSE;
	EXP_CMD := FALSE;
	GEN1_ON := FALSE;
	GEN2_ON := FALSE;
	ESS_ON := FALSE;
	BRK_toggle := 0;
	GEN1_toggle := 0;
	GEN2_toggle := 0;
	ESS_toggle := 0;
	Load_Cntr := 0;
	RUN_MIN := 0;
	MODE := 0;
	QG1_CMD := 0;
	QG2_CMD := 0;

END_PROGRAM

// Device/Application/POUs/Vijay
PROGRAM Vijay
VAR
	SUM: DINT := 1;
	INC: DINT := 0;
	//SET: BOOL;
	SET2: BOOL;
	T1_out: BOOL;
	T2_out: BOOL;
	Swtich_STAT: DINT := 0;
	Swtich_STAT1: DINT;
	SUM1: DINT;
	SET_R: BOOL;
	SET3: BOOL;
	RST1: INT;
	SUM2: DINT;
	T_ON: BOOL;
	TMR1: TON;
	TMR2: TON;
	RESET: RS;
	Out: BOOL;
	
	TMR3: TOF;
	T_OUT: BOOL;
	RST_B2: DINT := 0;
	SETRESET: SR;
	RST2_OUT: DINT;
	RS_1: RS;
	out16: DINT:= 0;
	Trig: BOOL:=1;
	RT_1: R_TRIG;
	TO_1: TOF;
	TRIG1: BOOL:=1;
	BOOL_AOS: BOOL;
	Amit: AO_STATE_ENUM;
	sample: DINT := 1;
	T1: DINT;
	UQ_Counter: CTU;
	LD_SHED: BOOL;
	CMD: BOOL;
	kCMD: BO_CMD_ENUM;
END_VAR

END_PROGRAM

// Device/Application/POUs/Timers
PROGRAM Timers
VAR
	STRT: BOOL := 1;
	TMRs: TON;
	TMR1: TON;
	STRT_2: BOOL := 1;
	T2_ET: TIME;
	MIN_RST: R_TRIG;
	TMR_SYS: BOOL := 0;
END_VAR

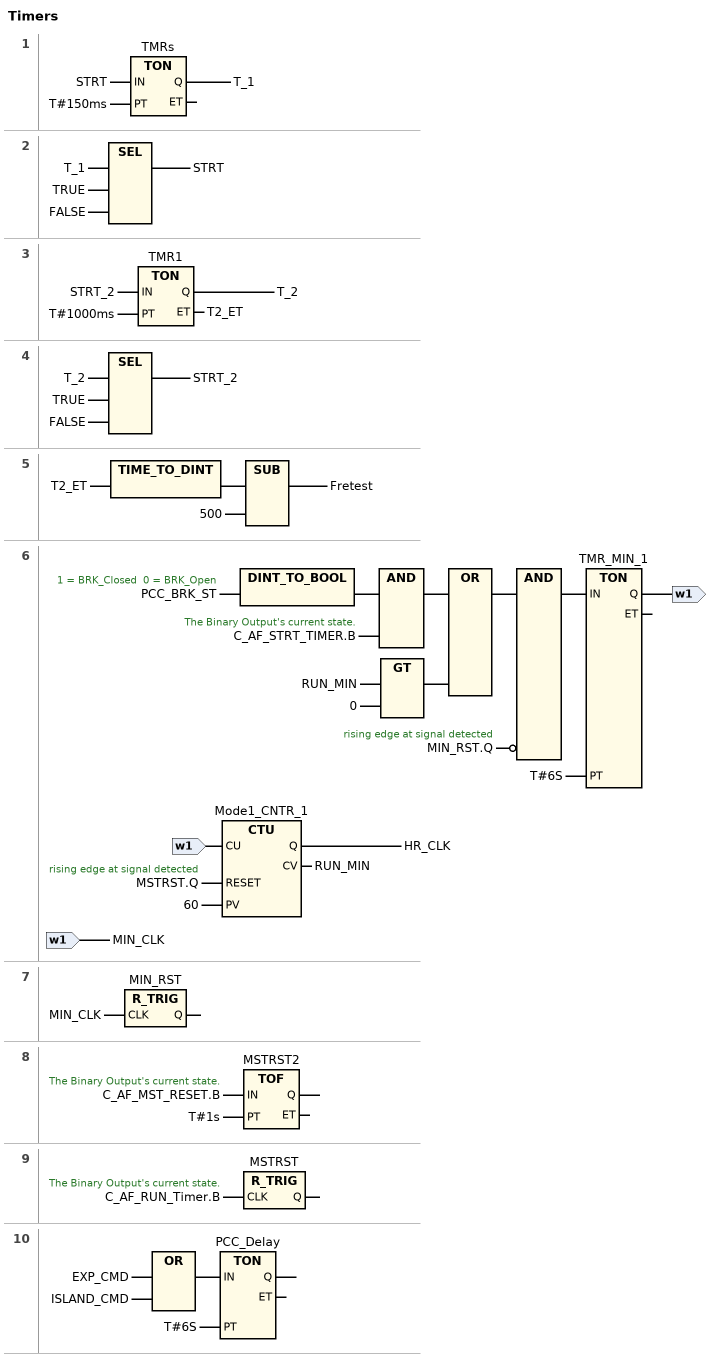
// NETWORK 1
TMRs(IN := STRT, PT := T#150ms); // TON
T_1 := TMRs.Q;

// NETWORK 2
STRT := SEL(T_1, TRUE, FALSE);

// NETWORK 3
TMR1(IN := STRT_2, PT := T#1000ms, ET => T2_ET); // TON
T_2 := TMR1.Q;

// NETWORK 4
STRT_2 := SEL(T_2, TRUE, FALSE);

// NETWORK 5
Fretest := TIME_TO_DINT(T2_ET) - 500;

// NETWORK 6
//   PCC_BRK_ST: 1 = BRK_Closed 0 = BRK_Open
//   C_AF_STRT_TIMER.B: The Binary Output's current state.
//   MIN_RST.Q: rising edge at signal detected
//   MSTRST.Q: rising edge at signal detected
TMR_MIN_1(IN := (DINT_TO_BOOL(PCC_BRK_ST) AND C_AF_STRT_TIMER.B OR RUN_MIN > 0) AND NOT MIN_RST.Q, PT := T#6S); // TON
Mode1_CNTR_1(CU := TMR_MIN_1.Q, RESET := MSTRST.Q, PV := 60, CV => RUN_MIN); // CTU
HR_CLK := Mode1_CNTR_1.Q;
MIN_CLK := TMR_MIN_1.Q;

// NETWORK 7
MIN_RST(CLK := MIN_CLK); // R_TRIG

// NETWORK 8
//   C_AF_MST_RESET.B: The Binary Output's current state.
MSTRST2(IN := C_AF_MST_RESET.B, PT := T#1s); // TOF

// NETWORK 9
//   C_AF_RUN_Timer.B: The Binary Output's current state.
MSTRST(CLK := C_AF_RUN_Timer.B); // R_TRIG

// NETWORK 10
PCC_Delay(IN := EXP_CMD OR ISLAND_CMD, PT := T#6S); // TON

END_PROGRAM

// Device/Application/POUs/Tasks_10ms
PROGRAM Tasks_10ms
VAR
END_VAR

vijay();

END_PROGRAM

// Device/Application/POUs/Tasks_50ms
PROGRAM Tasks_50ms
VAR
END_VAR

TIMER_ST();
//Timers();
//C_RUN_MIN(I :=RUN_MIN);

END_PROGRAM

// Device/Application/POUs/TIMER_ST
PROGRAM TIMER_ST
VAR
	Trig2: BOOL := 0;
	a: INT;
	b: INT;
	test: INT := 0;
END_VAR

AO_TGL_1(IN := Trig , PT := T#200MS); // IOP triger for SMP AO's
AO_TGL_2(IN := Trig2 , PT := T#200MS);

IF AO_TGL_1.Q THEN
	Trig2 := 1;
	Trig := 0;
END_IF

 
 IF AO_TGL_2.Q THEN
	 Trig := 1;
	 Trig2 := 0;
 END_IF
 IF Trig = 0 AND (Trig3<=2) THEN
	 Trig3:= Trig3+1;
	 ELSE
	 Trig3:=0;
 END_IF
IF Trig3<2 THEN
Trig4  := FALSE ;
ELSE
Trig4 :=TRUE;
END_IF 
//test := test+1;

END_PROGRAM

// Device/Application/POUs/Tasks_100ms
PROGRAM Tasks_100ms
VAR
END_VAR

//SMP_OUTPUTS();
//POU_RESET();
//VDC();

//PCC_CNTL();
//SMP_Csys_var_AI();
//SMP_Csys_var_AO();

END_PROGRAM

// Device/Application/POUs/SMP_OUTPUTS
PROGRAM SMP_OUTPUTS
VAR
END_VAR

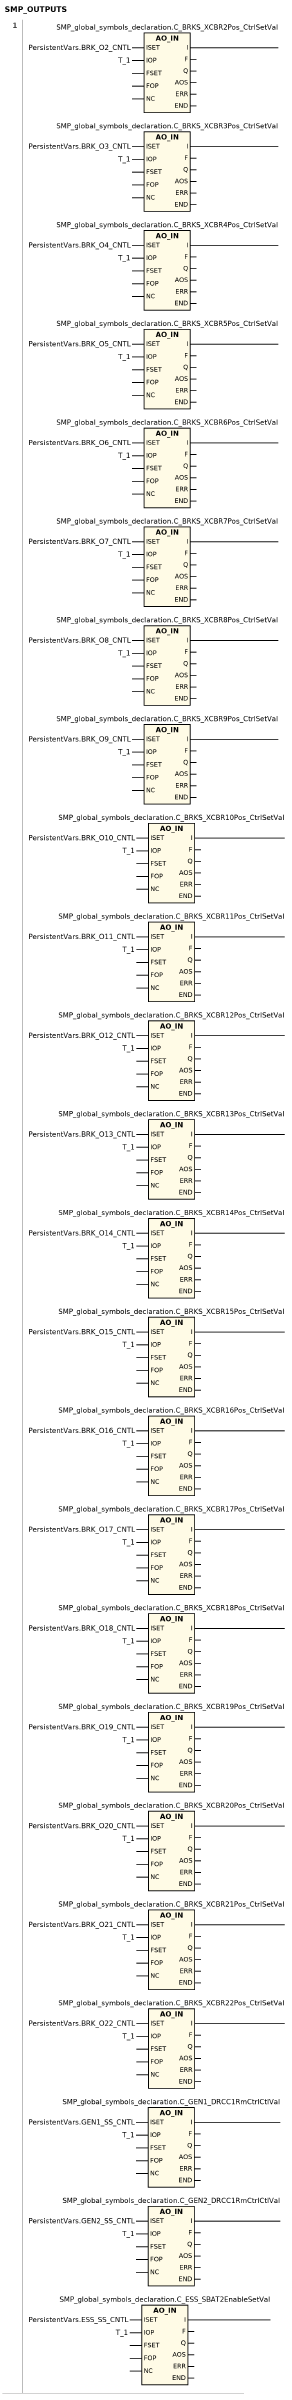
// NETWORK 1
//   SMP_global_symbols_declaration.C_BRKS_XCBR10Pos_CtrlSetVal: Consumed Ao
SMP_global_symbols_declaration.C_BRKS_XCBR2Pos_CtrlSetVal(ISET := PersistentVars.BRK_O2_CNTL, IOP := T_1); // AO_IN
SMP_global_symbols_declaration.C_BRKS_XCBR3Pos_CtrlSetVal(ISET := PersistentVars.BRK_O3_CNTL, IOP := T_1); // AO_IN
SMP_global_symbols_declaration.C_BRKS_XCBR4Pos_CtrlSetVal(ISET := PersistentVars.BRK_O4_CNTL, IOP := T_1); // AO_IN
SMP_global_symbols_declaration.C_BRKS_XCBR5Pos_CtrlSetVal(ISET := PersistentVars.BRK_O5_CNTL, IOP := T_1); // AO_IN
SMP_global_symbols_declaration.C_BRKS_XCBR6Pos_CtrlSetVal(ISET := PersistentVars.BRK_O6_CNTL, IOP := T_1); // AO_IN
SMP_global_symbols_declaration.C_BRKS_XCBR7Pos_CtrlSetVal(ISET := PersistentVars.BRK_O7_CNTL, IOP := T_1); // AO_IN
SMP_global_symbols_declaration.C_BRKS_XCBR8Pos_CtrlSetVal(ISET := PersistentVars.BRK_O8_CNTL, IOP := T_1); // AO_IN
SMP_global_symbols_declaration.C_BRKS_XCBR9Pos_CtrlSetVal(ISET := PersistentVars.BRK_O9_CNTL, IOP := T_1); // AO_IN
SMP_global_symbols_declaration.C_BRKS_XCBR10Pos_CtrlSetVal(ISET := PersistentVars.BRK_O10_CNTL, IOP := T_1); // AO_IN
SMP_global_symbols_declaration.C_BRKS_XCBR11Pos_CtrlSetVal(ISET := PersistentVars.BRK_O11_CNTL, IOP := T_1); // AO_IN
SMP_global_symbols_declaration.C_BRKS_XCBR12Pos_CtrlSetVal(ISET := PersistentVars.BRK_O12_CNTL, IOP := T_1); // AO_IN
SMP_global_symbols_declaration.C_BRKS_XCBR13Pos_CtrlSetVal(ISET := PersistentVars.BRK_O13_CNTL, IOP := T_1); // AO_IN
SMP_global_symbols_declaration.C_BRKS_XCBR14Pos_CtrlSetVal(ISET := PersistentVars.BRK_O14_CNTL, IOP := T_1); // AO_IN
SMP_global_symbols_declaration.C_BRKS_XCBR15Pos_CtrlSetVal(ISET := PersistentVars.BRK_O15_CNTL, IOP := T_1); // AO_IN
SMP_global_symbols_declaration.C_BRKS_XCBR16Pos_CtrlSetVal(ISET := PersistentVars.BRK_O16_CNTL, IOP := T_1); // AO_IN
SMP_global_symbols_declaration.C_BRKS_XCBR17Pos_CtrlSetVal(ISET := PersistentVars.BRK_O17_CNTL, IOP := T_1); // AO_IN
SMP_global_symbols_declaration.C_BRKS_XCBR18Pos_CtrlSetVal(ISET := PersistentVars.BRK_O18_CNTL, IOP := T_1); // AO_IN
SMP_global_symbols_declaration.C_BRKS_XCBR19Pos_CtrlSetVal(ISET := PersistentVars.BRK_O19_CNTL, IOP := T_1); // AO_IN
SMP_global_symbols_declaration.C_BRKS_XCBR20Pos_CtrlSetVal(ISET := PersistentVars.BRK_O20_CNTL, IOP := T_1); // AO_IN
SMP_global_symbols_declaration.C_BRKS_XCBR21Pos_CtrlSetVal(ISET := PersistentVars.BRK_O21_CNTL, IOP := T_1); // AO_IN
SMP_global_symbols_declaration.C_BRKS_XCBR22Pos_CtrlSetVal(ISET := PersistentVars.BRK_O22_CNTL, IOP := T_1); // AO_IN
SMP_global_symbols_declaration.C_GEN1_DRCC1RmCtrlCtlVal(ISET := PersistentVars.GEN1_SS_CNTL, IOP := T_1); // AO_IN
SMP_global_symbols_declaration.C_GEN2_DRCC1RmCtrlCtlVal(ISET := PersistentVars.GEN2_SS_CNTL, IOP := T_1); // AO_IN
SMP_global_symbols_declaration.C_ESS_SBAT2EnableSetVal(ISET := PersistentVars.ESS_SS_CNTL, IOP := T_1); // AO_IN

END_PROGRAM

// Device/Application/POUs/VDC
PROGRAM VDC
VAR
END_VAR

// ----Generator1 1MVA---//
F_G1_L := 59.5;
F_G1_H := 60.5;
V_G1_L := 0.95;
V_G1_H := 1.05;
//-----------------------//

//------Generator2 4MVA---//
F_G2_L := 59.5;
F_G2_H := 60.5;
V_G2_L := 0.95;
V_G2_H := 1.05;
//-----------------------//

//-------PV 3MW-----------//
F_PV_L := 59.5;
F_PV_H := 60.5;
V_PV_L := 0.95;
V_PV_H := 1.05;
//-----------------------//

//-----------S 4MW---------//
F_ES_L := 59.5;
F_ES_H := 60.5;
F_ES_L := 0.95;
F_ES_H := 1.05;
//-----------------------//

//---------Load------------//
F_L9_L := 59.5;
F_L9_H := 1.05;
F_L10_L := 59.5;
F_L10_H := 1.05;
F_L11_L := 59.5;
F_L11_H := 1.05;
F_L15_L := 59.5;
F_L15_H := 1.05;
F_L16_L := 59.5;
F_L16_H := 1.05;
F_L20_L := 59.5;
F_L20_H := 1.05;

V_L9_L := 0.95;
V_L9_H := 1.05;
V_L10_L := 0.95;
V_L10_H := 1.05;
V_L11_L := 0.95;
V_L11_H := 1.05;
V_L15_L := 0.95;
V_L15_H := 1.05;
V_L16_L := 0.95;
V_L16_H := 1.05;
V_L20_L := 0.95;
V_L20_H := 1.05;
//-----------------------//

//-----Base Load Frequency/Voltage limit----//
F_BL_L := 59.5;
F_BL_H := 60.5;
V_BL_L := 0.95;
V_BL_H := 1.05;
//---------------------------------//

//---------------------------------------------Total Microgrid Load-----------------------------------------------------------//
//This is the SUM of breakers 2 to 22//
//Adding breaker1(PCC breaker with an -ve sign gives a total load in the Microgrid)//
(*
PTL := P_R5+P_R9+P_R10+P_R11+P_R14+P_R15+P_R16+P_R18+P_R19+P_R20+P_R21+P_R22;//P_R2+P_R3+P_R4++P_R6+P_R12+P_R13P_R17+P_R7+P_R8
QTL := Q_R5+Q_R9+Q_R10+Q_R11+Q_R14+Q_R15+Q_R16+Q_R18+Q_R19+Q_R20+Q_R21+Q_R22;//Q_R2+Q_R3+Q_R4++Q_R6+Q_R12Q_R13Q_R17+Q_R7+Q_R8
*)
 
PTL := C_PCC1_MMXU1TotWMag.F -P_R7 -P_R8 -P_R13 -P_R17;
QTL := C_PCC1_MMXU1TotVArMag.F -Q_R7 -Q_R8 -Q_R13 -Q_R17;

//---------------------------------------------------------------------------------------------------------------------------//

//------------MODE1 Load----------------------//
PTL_Mode1 := PTL - C_SOLAR_ZINV1TotWMag.F ; // Real Power from GRID- C_GEN1_MMXU1TotWMag.F - C_GEN2_MMXU1TotWMag.F - C_ESS_SBAT2TotWMag.F
QTL_Mode1 := QTL - C_ESS_SBAT2TotVArMag.F;    // Reactive Power from GRID
//-------------------------------------------//

//------------MODE2 Load----------------------//
(*
PTL_Mode2 := PTL + C_ESS_SBAT2TotWMag.F; // Real Power from ESS
QTL_Mode2 := QTL + C_ESS_SBAT2Cap_VARMag.F; // Reactive Power from ESS
*)

PTL_Mode2 := P_R2+P_R3+P_R4+P_R7+P_R8;
QTL_Mode2 := Q_R2+Q_R3+Q_R4+Q_R7+Q_R8;

//-------------------------------------------//


//----------Base Load of Microgrid----------//
MG_Base_P := C_AF_MG_Base_P.F;    //9;
MG_Base_Q := C_AF_MG_Base_Q.F;   //5;
//----------------------------------------//


//----------Application Selection-----------//
GRID_APP_SELECT:= 1;  //GRID Mode Export Application
ISLAND_APP_SELECT:= 1; //ISLAND Mode LOAD balancing Application
//----------------------------------------//

END_PROGRAM

// Device/Application/POUs/PCC_CNTL
PROGRAM PCC_CNTL
VAR
	PCC_BRK_ST1: R_TRIG;
	
	Force: BOOL := 0;
END_VAR

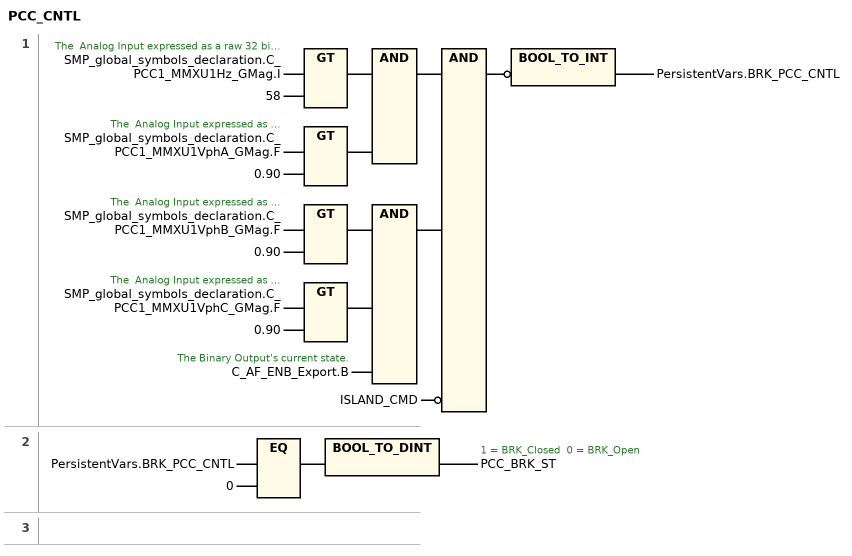
// NETWORK 1
//   SMP_global_symbols_declaration.C_PCC1_MMXU1Hz_GMag.I: The Analog Input expressed as a raw 32 bit signed integer.
//   SMP_global_symbols_declaration.C_PCC1_MMXU1VphA_GMag.F: The Analog Input expressed as a floating-point value.
//   SMP_global_symbols_declaration.C_PCC1_MMXU1VphB_GMag.F: The Analog Input expressed as a floating-point value.
//   SMP_global_symbols_declaration.C_PCC1_MMXU1VphC_GMag.F: The Analog Input expressed as a floating-point value.
//   C_AF_ENB_Export.B: The Binary Output's current state.
PersistentVars.BRK_PCC_CNTL := BOOL_TO_INT(NOT ((SMP_global_symbols_declaration.C_PCC1_MMXU1Hz_GMag.I > 58 AND SMP_global_symbols_declaration.C_PCC1_MMXU1VphA_GMag.F > 0.90) AND (SMP_global_symbols_declaration.C_PCC1_MMXU1VphB_GMag.F > 0.90 AND SMP_global_symbols_declaration.C_PCC1_MMXU1VphC_GMag.F > 0.90 AND C_AF_ENB_Export.B) AND NOT ISLAND_CMD));

// NETWORK 2
//   PCC_BRK_ST: 1 = BRK_Closed 0 = BRK_Open
PCC_BRK_ST := BOOL_TO_DINT(PersistentVars.BRK_PCC_CNTL = 0);

// NETWORK 3

END_PROGRAM

// Device/Application/POUs/SMP_Csys_var_AI
PROGRAM SMP_Csys_var_AI
VAR
END_VAR

P_R2 := C_BRKS_XCBR2TotWMag.F;
P_R3 := C_BRKS_XCBR3TotWMag.F;
P_R4 := C_BRKS_XCBR4TotWMag.F;
P_R5 := C_BRKS_XCBR5TotWMag.F;
P_R6 := C_BRKS_XCBR6TotWMag.F;
P_R7 := C_BRKS_XCBR7TotWMag.F;
P_R8 := C_BRKS_XCBR8TotWMag.F;
P_R9 := C_BRKS_XCBR9TotWMag.F;
P_R10 := C_BRKS_XCBR10TotWMag.F;
P_R11 := C_BRKS_XCBR11TotWMag.F;
P_R12 := C_BRKS_XCBR12TotWMag.F;
P_R13 := C_BRKS_XCBR13TotWMag.F;
P_R14 := C_BRKS_XCBR14TotWMag.F;
P_R15 := C_BRKS_XCBR15TotWMag.F;
P_R16 := C_BRKS_XCBR16TotWMag.F;
P_R17 := C_BRKS_XCBR17TotWMag.F;
P_R18 := C_BRKS_XCBR18TotWMag.F;
P_R19 := C_BRKS_XCBR19TotWMag.F;
P_R20 := C_BRKS_XCBR20TotWMag.F;
P_R21 := C_BRKS_XCBR21TotWMag.F;
P_R22 := C_BRKS_XCBR22TotWMag.F;

Q_R2 := C_BRKS_XCBR2TotVArMag.F;
Q_R3 := C_BRKS_XCBR3TotVArMag.F;
Q_R4 := C_BRKS_XCBR4TotVArMag.F;
Q_R5 := C_BRKS_XCBR5TotVArMag.F;
Q_R6 := C_BRKS_XCBR6TotVArMag.F;
Q_R7 := C_BRKS_XCBR7TotVArMag.F;
Q_R8 := C_BRKS_XCBR8TotVArMag.F;
Q_R9 := C_BRKS_XCBR9TotVArMag.F;
Q_R10 := C_BRKS_XCBR10TotVArMag.F;
//Q_R11 := C_BRKS_XCBR11TotVArMag.F;
Q_R12 := C_BRKS_XCBR12TotVArMag.F;
Q_R13 := C_BRKS_XCBR13TotVArMag.F;
Q_R14 := C_BRKS_XCBR14TotVArMag.F;
Q_R15 := C_BRKS_XCBR15TotVArMag.F;
Q_R16 := C_BRKS_XCBR16TotVArMag.F;
Q_R17 := C_BRKS_XCBR17TotVArMag.F;
Q_R18 := C_BRKS_XCBR18TotVArMag.F;
Q_R19 := C_BRKS_XCBR19TotVArMag.F;
Q_R20 := C_BRKS_XCBR20TotVArMag.F;
Q_R21 := C_BRKS_XCBR21TotVArMag.F;
Q_R22 := C_BRKS_XCBR22TotVArMag.F;	

//PPCC_G := C_PCC1_MMXU1TotWMag.F; // Real Power from GRID
//QPCC_G := C_PCC1_MMXU1TotVArMag.F; 	


Gen1_CapW := C_GEN1_MMXU1Cap_WMag.F;
Gen2_CapW := C_GEN2_MMXU1Cap_WMag.F;
Gen1_Capkvar := C_AF_GEN1_Cap_VARMag.F;//C_GEN1_MMXU1Cap_VARMag.F;
Gen2_Capkvar := C_AF_GEN2_Cap_VARMag.F;//C_GEN2_MMXU1Cap_VARMag.F;

END_PROGRAM

// Device/Application/POUs/SMP_Csys_var_AO
PROGRAM SMP_Csys_var_AO
VAR
END_VAR

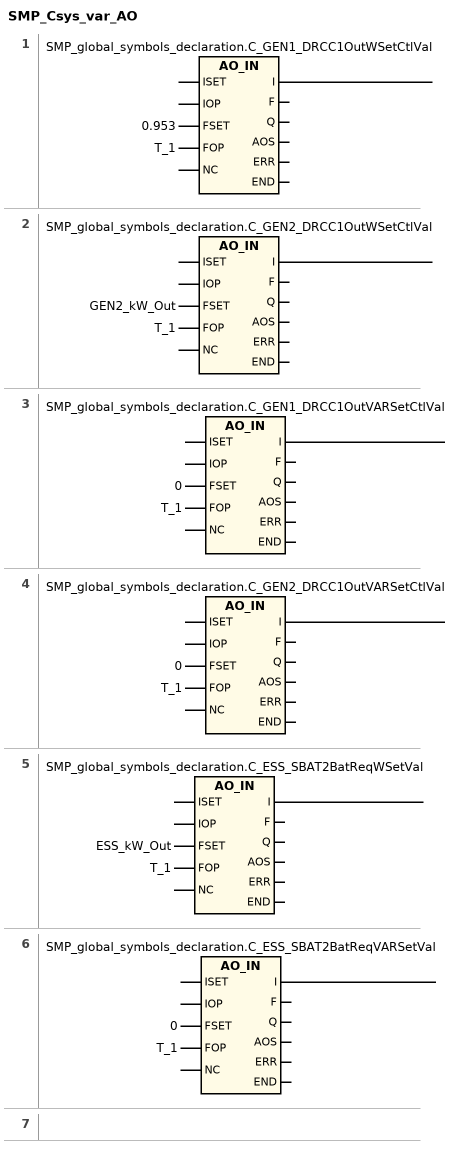
// NETWORK 1
SMP_global_symbols_declaration.C_GEN1_DRCC1OutWSetCtlVal(FSET := 0.953, FOP := T_1); // AO_IN

// NETWORK 2
SMP_global_symbols_declaration.C_GEN2_DRCC1OutWSetCtlVal(FSET := GEN2_kW_Out, FOP := T_1); // AO_IN

// NETWORK 3
SMP_global_symbols_declaration.C_GEN1_DRCC1OutVARSetCtlVal(FSET := 0, FOP := T_1); // AO_IN

// NETWORK 4
SMP_global_symbols_declaration.C_GEN2_DRCC1OutVARSetCtlVal(FSET := 0, FOP := T_1); // AO_IN

// NETWORK 5
SMP_global_symbols_declaration.C_ESS_SBAT2BatReqWSetVal(FSET := ESS_kW_Out, FOP := T_1); // AO_IN

// NETWORK 6
SMP_global_symbols_declaration.C_ESS_SBAT2BatReqVARSetVal(FSET := 0, FOP := T_1); // AO_IN

// NETWORK 7

END_PROGRAM

// Device/Application/POUs/Task_300ms
PROGRAM Task_300ms
VAR
END_VAR

//SMP_AO();
//MICROGRID_MODES();
//PCC_CNTL();
//BRK_CNTL();
//LOAD_Balance();
//SOC_MNGT();
//SMP_Csys_var_AO();

END_PROGRAM

// Device/Application/POUs/SMP_AO
PROGRAM SMP_AO
VAR
END_VAR


IF EXP_CMD THEN
SMP_global_symbols_declaration.C_GEN1_DRCC1OutWSetCtlVal(FSET := GEN1_kW_Out , FOP :=  Trig4);
SMP_global_symbols_declaration.C_GEN2_DRCC1OutWSetCtlVal(FSET := GEN2_kW_Out , FOP :=  Trig4);
SMP_global_symbols_declaration.C_ESS_SBAT2BatReqWSetVal(FSET := ESS_kW_Out , FOP := Trig);
SMP_global_symbols_declaration.C_GEN1_DRCC1OutVARSetCtlVal(FSET := QG1_CMD , FOP :=  Trig4);
SMP_global_symbols_declaration.C_GEN2_DRCC1OutVARSetCtlVal(FSET := QG2_CMD , FOP :=  Trig4);
SMP_global_symbols_declaration.C_ESS_SBAT2BatReqVARSetVal(FSET := ESS_kVAr_Out , FOP :=  Trig4);
END_IF

IF ISLAND_CMD THEN
SMP_global_symbols_declaration.C_GEN1_DRCC1OutWSetCtlVal(FSET := PG1_CMD , FOP :=  Trig4);
SMP_global_symbols_declaration.C_GEN2_DRCC1OutWSetCtlVal(FSET := PG2_CMD , FOP :=  Trig4);
SMP_global_symbols_declaration.C_GEN1_DRCC1OutVARSetCtlVal(FSET := QG1_CMD , FOP :=  Trig4);
SMP_global_symbols_declaration.C_GEN2_DRCC1OutVARSetCtlVal(FSET := QG2_CMD , FOP :=  Trig4);
//SMP_global_symbols_declaration.C_ESS_SBAT2BatReqVARSetVal(FSET := ESS_kVAr_Out , FOP :=  Trig4);

END_IF
//SMP_global_symbols_declaration.C_GEN1_DRCC1OutWSetCtlVal.END
//SMP_global_symbols_declaration.C_GEN1_DRCC1OutWSetCtlVal.ERR
//SMP_global_symbols_declaration.C_GEN2_DRCC1OutWSetCtlVal.END
//SMP_global_symbols_declaration.C_GEN2_DRCC1OutWSetCtlVal.ERR	
//SMP_global_symbols_declaration.C_ESS_SBAT2BatReqWSetVal.END
//SMP_global_symbols_declaration.C_ESS_SBAT2BatReqWSetVal.ERR

END_PROGRAM

// Device/Application/POUs/MICROGRID_MODES
PROGRAM MICROGRID_MODES
VAR
END_VAR

IF PCC_BRK_ST = 1 THEN
	MODE := 1;  //GRID
END_IF  

IF ISLAND_CMD = 1 THEN  //PCC_BRK_ST
	MODE := 2;  //ISLAND
END_IF

MICROGRID_Apps();

END_PROGRAM

// Device/Application/POUs/MICROGRID_Apps
PROGRAM MICROGRID_Apps
VAR
END_VAR

IF MODE = 1 THEN
	CASE GRID_APP_SELECT  OF   // APQ_SELECT := (Value from VTD)
	1:POU_EXPORT();
	Q_Export();
//	2:POU_DR()
//	3:POU_FR()	
	END_CASE
END_IF

IF MODE = 2 THEN
	CASE ISLAND_APP_SELECT  OF   // APQ_SELECT := (Value from VTD)
	1:LOAD_Balance();
//	2:POU_DR()
//	3:POU_FR()	
	END_CASE
END_IF

END_PROGRAM

// Device/Application/POUs/POU_EXPORT
PROGRAM POU_EXPORT
VAR

	Offset: REAL := 0.05;
	Freq_Err: REAL := 0;
	ESS_kW_Out1: REAL :=0; 
END_VAR

Freq_Err := SPS_SELG_METYMMXU2HzInstMag.F - 60.0 - Offset;

PV_kW_Out := (((SPS_ADAM1_ADAM_AI_5.F - 32767) / 32767 * 10 / 251 / 2.5 * 43000) * (((SPS_ADAM1_ADAM_AI_3.F- 32767) / 32767 * 10 / 251 - 0.004) / 0.02 * 150 * 1.414213) / 1000)-0.13;


//ESS_kVAr_Out := ESS_kVAr_Out+1;

IF SPS_GEN1_METMMXU1TotWInstMag.F > 10.0 THEN
	IF (Freq_Err > 0.0) THEN
		ESS_kW_Out1 := ESS_kW_Out1 + 1;
		ELSE
		ESS_kW_Out1 := ESS_kW_Out1 - 1;
	END_IF
	ELSE
	ESS_kW_Out1 := 0;
END_IF





SMP_global_symbols_declaration.SPS_PCS_INV1_FB2_POWDEL_INS(FSET := ESS_kW_Out1 , FOP :=  Trig4);
SMP_global_symbols_declaration.SPS_PCS_INV1_FB3_POWDEL_INS(FSET := ESS_kVAr_Out , FOP :=  Trig4);

END_PROGRAM

// Device/Application/POUs/Q_Export
PROGRAM Q_Export
VAR
	PCC_Q_EXP: REAL := 0;
	MG_kVAr_Out: REAL := 0;
	INT_ERR_Q: REAL := 0;
	GEN1_Q_CAP: REAL := 0;
	G1QCap: REAL := 0.6;
	GEN2_Q_CAP: REAL := 0;
	G2QCap: REAL := 2.4;
	PPCC_Q_CMD: REAL := 0;
	ERR_T_Q: REAL := 0;
	INT_ERR_A: REAL := 0;
	KI_Q: REAL := 0;
	KP_Q: REAL := 0;
	INT_ERR_LIM: REAL := 150.0;
	INT_ERR_LIML: REAL := -150.0;
	MG_kVAr_Bal2: REAL := 0;
	MG_kVAr_Bal3: REAL := 0;
	BAT_CAP_Q: REAL := 0;
END_VAR



//-----------------------------------------------------Q calculation-----------------------------------------------//
GEN1_Q_CAP := 20.0; //C_AF_GEN1_Cap_VARMag.F
BAT_CAP_Q := 20.0;
KI_Q := 0.0011;
KP_Q := 0.21;
	IF ABS(SPS_GEN1_METMMXU1TotVArInstMag.F) > 0.0 THEN
		ERR_T_Q := PPCC_Q_CMD + SPS_GEN1_METMMXU1TotVArInstMag.F; // PCCC_Q_CMD may be based on timer
		INT_ERR_A := ERR_T_Q + INT_ERR_Q;
		
		IF INT_ERR_A >= INT_ERR_LIM THEN
			INT_ERR_Q := INT_ERR_LIM;
		END_IF
		IF INT_ERR_A <= INT_ERR_LIML THEN
			INT_ERR_Q := INT_ERR_LIML;
		END_IF		
		
		IF (INT_ERR_A <=  INT_ERR_LIM)  AND  (INT_ERR_A >=  INT_ERR_LIML)  THEN
			INT_ERR_Q := INT_ERR_LIM;
		END_IF		
	
	ESS_kVAr_Out := SPS_GEN1_METMMXU1TotVArInstMag.F + INT_ERR_Q*KI_Q + ERR_T_Q*KP_Q;
	
	IF ESS_kVAr_Out > 20.0 THEN
		ESS_kVAr_Out := 20.0;
	END_IF
	IF ESS_kVAr_Out < -5.0 THEN
		ESS_kVAr_Out := -5.0;
	END_IF
	
	IF (ESS_kVAr_Out > (BAT_CAP_Q)) THEN       //C_AF_GEN1_Cap_WMag.F
			ESS_kVAr_Out := (BAT_CAP_Q);         //C_GEN1_MMXU1Cap_WMag.FC_AF_GEN1_Cap_WMag.F
	END_IF
(*		
	MG_kVAr_Bal2 := MG_kVAr_Out - GEN1_kVAr_Out - GEN2_kVAr_Out;		
		
		IF MG_kVAr_Bal2 > 0 THEN
			MG_kVAr_Bal3 := MG_kVAr_Bal2;
			ELSE
			MG_kVAr_Bal3 := 0.0;	
		END_IF
		IF MG_kVAr_Bal3 > 0 THEN
			IF MG_kVAr_Bal3 > (BAT_CAP_Q) THEN  // Define Bat_cap_Q based on ESS_KW command
				ESS_kVAr_Out := ((1.0)*(BAT_CAP_Q)); 
				ELSE
				ESS_kVAr_Out := (1.0)*MG_kVAr_Bal3;
			END_IF
		END_IF
		
		IF MG_kVAr_Out <= 0 THEN
			IF MG_kVAr_Out < ((-1.0)*BAT_CAP_Q) THEN 
				ESS_kVAr_Out := (-1*BAT_CAP_Q);
			END_IF
			IF (MG_kVAr_Out <=0.0) AND (MG_kVAr_Out >= ((-1.0)*(BAT_CAP_Q)))  THEN
				ESS_kVAr_Out := (1.0)*MG_kVAr_Out;
			END_IF
		END_IF

	QG1_CMD := GEN1_kVAr_Out;
	QG2_CMD := GEN2_kVAr_Out;

*)

	END_IF
	//-----------------------------------------//

END_PROGRAM

// Device/Application/POUs/LOAD_Balance
PROGRAM LOAD_Balance
VAR
	ERR_P: REAL := 0;
	INT_ERR_P: REAL := 0;
	KI_I: REAL := 0;
	KP_I: REAL := 0;
	PTL_MD2_COR: REAL :=0;
	F_I: REAL := 0;
	ERR_Q: REAL := 0;
	INT_ERR_Q: REAL := 0;
	KI_IQ: REAL := 0;
	KP_IQ: REAL := 0;
	QTL_MD2_COR: REAL := 0;
	V_I: LREAL := 0;
END_VAR

Load_Shed();

//--------------PESS_CMD-------------------//
(*
F := F_BL_H - ((PTL_Mode2 / (MG_Base_P+0.001)) * (F_BL_H - F_BL_L));
IF F < F_G1_H THEN
PG1_CMD := ((F_G1_H -F ) / (F_G1_H - F_G1_L))* (Gen1_CapW);
END_IF
IF F < F_G2_H THEN
PG2_CMD := ((F_G2_H - F) / (F_G2_H - F_G2_L))* (Gen2_CapW);
END_IF
*)
//--------------PESS_CMD-------------------//

IF ISLAND_CMD THEN

F_I := F_BL_H + (((PTL_Mode2 + PTL_MD2_COR) / (MG_Base_P)) * (F_BL_H - F_BL_L));
IF F_I < 59.5 THEN
	F := 59.5;
	ELSIF F_I > 60.5 THEN
		F := 60.5;
END_IF

IF (F_I < 60.5) AND (F_I > 59.5) THEN 
		F := F_I;
END_IF		
		
IF F < F_G1_H THEN
PG1_CMD := ((F_G1_H -F ) / (F_G1_H - F_G1_L))* (C_AF_GEN1_Cap_WMag.F);   //Gen1_CapW=1
END_IF
IF F < F_G2_H THEN
PG2_CMD := ((F_G2_H - F) / (F_G2_H - F_G2_L))* (C_AF_GEN2_Cap_WMag.F);   //Gen2_CapW=4
END_IF

	ERR_P := P_R13; 
	INT_ERR_P := ERR_P + INT_ERR_P;
	KI_I := 0.06; // := C_AF_KI_I.F ;
	KP_I := 0.06;  //C_AF_KP_I.F
	PTL_MD2_COR := ERR_P*KP_I  + INT_ERR_P*KI_I  ;
	
END_IF




//----------------------------------------//


//------------------QESS_CMD--------------//
V := V_BL_H + (((QTL_Mode2 - QTL_MD2_COR)/ (MG_Base_Q+0.0001)) * (V_BL_H - V_BL_L));
IF V_I < 0.95 THEN
	V := 0.95;
	ELSIF V_I > 1.05 THEN
		V := 1.05;
END_IF
IF (V_I < 0.95) AND (V_I > 1.05) THEN 
		V := V_I;
END_IF

IF V < 1.0 THEN
QG1_CMD_A := ((1.0 - V) / (1.0 - V_G1_L))* (Gen1_Capkvar);
END_IF

IF V > 1.0 THEN
QG1_CMD_A := ((V - 1.0) / (V_G1_H - 1.0))* (Gen1_Capkvar);
END_IF

IF QG1_CMD_A > Gen1_Capkvar THEN
	QG1_CMD := Gen1_Capkvar;
END_IF

IF QG1_CMD_A < (-1*Gen1_Capkvar) THEN
	QG1_CMD := (-1*Gen1_Capkvar);
END_IF 

IF (QG1_CMD_A < Gen1_Capkvar) AND (QG1_CMD_A > (-1*Gen1_Capkvar))  THEN
	QG1_CMD := QG1_CMD_A;
END_IF 


(*
IF V < V_G2_H THEN
QG2_CMD_A := ((V_G2_H - V) / (V_G2_H - V_G2_L))* (Gen2_Capkvar);
END_IF
IF QG2_CMD_A > C_AF_GEN2_Cap_VARMag.F THEN
	QG2_CMD := C_AF_GEN2_Cap_VARMag.F;
ELSE
	QG2_CMD := QG2_CMD_A;
END_IF
*)
IF V < 1.0 THEN
QG2_CMD_A := ((1.0 - V) / (1.0 - V_G2_L))* (Gen2_Capkvar);
END_IF

IF V > 1.0 THEN
QG2_CMD_A := ((V - 1.0) / (V_G2_H - 1.0))* (Gen2_Capkvar);
END_IF

IF QG2_CMD_A > Gen2_Capkvar THEN
	QG2_CMD := Gen2_Capkvar;
END_IF

IF QG2_CMD_A < (-1*Gen2_Capkvar) THEN
	QG2_CMD := (-1*Gen2_Capkvar);
END_IF 

IF (QG2_CMD_A < Gen2_Capkvar) AND (QG2_CMD_A > (-1*Gen2_Capkvar))  THEN
	QG2_CMD := QG2_CMD_A;
END_IF 


//----------------------------------------//

END_PROGRAM

// Device/Application/POUs/Load_Shed
PROGRAM Load_Shed
VAR

	
END_VAR

IF (ISLAND_CMD) THEN
	I_Load_05 := 0;
	I_Load_09 := 0;
	I_Load_10 := 0;
	I_Load_11 := 0;
	I_Load_015 := 0;
	I_Load_016 := 0;
//	I_Load_020 := 0;

Load_Cntr := Load_Cntr+1;	
END_IF




IF Load_Cntr > 150 THEN
	I_Load_05 := 1;
END_IF
IF Load_Cntr > 200 THEN
	I_Load_09 := 1;
END_IF
IF Load_Cntr > 250 THEN
	I_Load_10 := 1;
END_IF
IF Load_Cntr > 300 THEN
	I_Load_11 := 1;
END_IF
IF Load_Cntr > 350 THEN
	I_Load_015 := 1;
END_IF
IF Load_Cntr > 400 THEN
	I_Load_016 := 1;
END_IF

IF Load_Cntr >= 450 THEN
	Load_Cntr := 450;
END_IF

(*

IF (PCC_BRK_ST = 0 AND I_Load_05 = 1 )THEN
	PersistentVars.BRK_O5_CNTL := 0;
END_IF

IF (PCC_BRK_ST = 0 AND I_Load_09 = 1 )THEN
	PersistentVars.BRK_O9_CNTL := 0;
END_IF

IF (PCC_BRK_ST = 0 AND I_Load_10 = 1 )THEN
	PersistentVars.BRK_O10_CNTL:= 0;
END_IF

IF (PCC_BRK_ST = 0 AND I_Load_11 = 1 )THEN
	PersistentVars.BRK_O11_CNTL := 0;
END_IF

IF (PCC_BRK_ST = 0 AND I_Load_014 = 1 )THEN
	PersistentVars.BRK_O14_CNTL := 0;
END_IF

IF (PCC_BRK_ST = 0 AND I_Load_015 = 1 )THEN
	PersistentVars.BRK_O15_CNTL := 0;
END_IF

IF (PCC_BRK_ST = 0 AND I_Load_016 = 1 )THEN
	PersistentVars.BRK_O16_CNTL := 0;
END_IF

IF (PCC_BRK_ST = 0 AND I_Load_020 = 1 )THEN
	PersistentVars.BRK_O20_CNTL := 0;
END_IF

*)
/* Comment*/

END_PROGRAM

// Device/Application/POUs/SOC_MNGT
PROGRAM SOC_MNGT
VAR
END_VAR

//--------Export Mode---------------//
IF EXP_CMD = 1 THEN

	IF C_ESS_SBAT2SoCMag.F < 6.0 THEN
		BAT_CAP := C_AF_ESS_SBAT2Cap_WMag.F*(C_ESS_SBAT2SoCMag.F - 5);//C_ESS_SBAT2Cap_WMag.F
	END_IF
	IF C_ESS_SBAT2SoCMag.F < C_AF_MIN_SOC.F THEN //5.0
		BAT_CAP := 0;
	END_IF
	IF C_ESS_SBAT2SoCMag.F > 6.0 AND  C_ESS_SBAT2SoCMag.F < 95.0 THEN
		BAT_CAP := C_AF_ESS_SBAT2Cap_WMag.F;//C_ESS_SBAT2Cap_WMag.F
	END_IF
		
	IF C_ESS_SBAT2SoCMag.F > 95.0 THEN
		BAT_CAP := C_AF_ESS_SBAT2Cap_WMag.F*(C_AF_MAX_SOC.F - C_ESS_SBAT2SoCMag.F);  //96C_ESS_SBAT2Cap_WMag.F
	END_IF
	IF C_ESS_SBAT2SoCMag.F > C_AF_MAX_SOC.F THEN   //96.0
		BAT_CAP := 0;
	END_IF
		
	IF C_ESS_SBAT2SoCMag.F < 50.0 AND PPCC_CMD = 0 THEN
		ESS_kW_Out := 1.0;
	END_IF
	
	IF C_ESS_SBAT2SoCMag.F > 50.0 AND PPCC_CMD = 0 THEN
		ESS_kW_Out := -1.0;
	END_IF
	
END_IF

//----------------------------------//



IF ISLAND_APP_SELECT = 1 THEN
//--------Island Mode---------------//
//----------------------------------//

END_IF

END_PROGRAM

// GetNumberProperty
// This function has been automatically generated from the project information.
{attribute 'signature_flag' := '1073741824'}
{attribute 'register_in_runtime'}
FUNCTION GetNumberProperty : DINT
VAR_INPUT
	stKey: WSTRING;
END_VAR

GetNumberProperty := 0;

END_FUNCTION

// GetBooleanProperty
// This function has been automatically generated from the project information.
{attribute 'signature_flag' := '1073741824'}
{attribute 'register_in_runtime'}
FUNCTION GetBooleanProperty : BOOL
VAR_INPUT
	stKey: WSTRING;
END_VAR

IF stKey = "Released" THEN
	GetBooleanProperty := FALSE;
ELSE
	GetBooleanProperty := FALSE;
END_IF

END_FUNCTION

// GetCompany
// This function has been automatically generated from the project information.
{attribute 'signature_flag' := '1073741824'}
{attribute 'register_in_runtime'}
FUNCTION GetCompany : WSTRING
VAR_INPUT
	
END_VAR

GetCompany := "Cooper Power Systems LLC";

END_FUNCTION

// GetTitle
// This function has been automatically generated from the project information.
{attribute 'signature_flag' := '1073741824'}
{attribute 'register_in_runtime'}
FUNCTION GetTitle : WSTRING
VAR_INPUT
	
END_VAR

GetTitle := "CoDeSys Project";

END_FUNCTION

// GetVersionProperty
// This function has been automatically generated from the project information.
{attribute 'signature_flag' := '1073741824'}
{attribute 'register_in_runtime'}
FUNCTION GetVersionProperty : VERSION
VAR_INPUT
	stKey: WSTRING;
END_VAR

IF stKey = "Version" THEN
	GetVersionProperty.uiMajor := 1;
	GetVersionProperty.uiMinor := 0;
	GetVersionProperty.uiServicePack := 0;
	GetVersionProperty.uiPatch := 0;
ELSE
	GetVersionProperty.uiMajor := 0;
	GetVersionProperty.uiMinor := 0;
	GetVersionProperty.uiServicePack := 0;
	GetVersionProperty.uiPatch := 0;
END_IF

END_FUNCTION

// GetVersion
// This function has been automatically generated from the project information.
{attribute 'signature_flag' := '1073741824'}
{attribute 'register_in_runtime'}
FUNCTION GetVersion : VERSION
VAR_INPUT
	
END_VAR

GetVersion.uiMajor := 1;
GetVersion.uiMinor := 0;
GetVersion.uiServicePack := 0;
GetVersion.uiPatch := 0;

END_FUNCTION

// GetTextProperty
// This function has been automatically generated from the project information.
{attribute 'signature_flag' := '1073741824'}
{attribute 'register_in_runtime'}
FUNCTION GetTextProperty : WSTRING
VAR_INPUT
	stKey: WSTRING;
END_VAR

IF stKey = "Author" THEN
	GetTextProperty := "Cooper Power Systems";
ELSIF stKey = "Company" THEN
	GetTextProperty := "Cooper Power Systems LLC";
ELSIF stKey = "Description" THEN
	GetTextProperty := "Sample Project";
ELSIF stKey = "Project" THEN
	GetTextProperty := "CoDeSysProj";
ELSIF stKey = "Title" THEN
	GetTextProperty := "CoDeSys Project";
ELSIF stKey = "Version string" THEN
	GetTextProperty := "";
ELSE
	GetTextProperty := "";
END_IF

END_FUNCTION

// Device/Application/POUs/PCC_PROTECT
PROGRAM PCC_PROTECT
VAR
END_VAR

END_PROGRAM
